// TIA Portal project "GoodBeer_V1" (V16)

(* hardware
DEVICE "Станция S7-1200_1"  S7-1200 Station
   slot 0: "Rack_0"  S7-1200 Rack  Rack  V1.0
   slot 1: "PLC"  CPU 1214C DC/DC/Rly  6ES7 214-1HG40-0XB0  V4.2
   slot 2: "DI 16x24VDC_1"  6ES7 221-1BH32-0XB0  V2.0
   slot 3: "DQ 16xRelay_1"  SM 1222 DQ16 x relay  6ES7 222-1HH32-0XB0  V2.0
   slot 4: "DQ 8xRelay_1"  SM 1222 DQ8 x relay  6ES7 222-1HF32-0XB0  V2.0
   slot 5: "AI 8xRTD_1"  SM 1231 AI8 x RTD  6ES7 231-5PF32-0XB0  V2.0
   slot 6: "AI 8x13 бит_1"  6ES7 231-4HF32-0XB0  V2.0
   slot 7: "AQ 4x14 бит_1"  6ES7 232-4HD32-0XB0  V2.0
   slot 8: "AQ 4x14 бит_2"  6ES7 232-4HD32-0XB0  V2.0
*)

// ===== PLC "PLC"  CPU 1214C DC/DC/Rly =====

VAR_GLOBAL   // PLC tag table "Стандартная таблица переменных"
   "Возврат(1)" AT %M10.6 : Bool;
   "Клавиша Стопа на экране" AT %M202.1 : Bool;
   "клавиша циркуляции" AT %M279.1 : Bool;
   "Циркуляция" AT %M247.2 : Bool;
   "Клапана  в автомат" AT %M38.1 : Bool;
   "mm3" AT %M38.3 : Bool;
   "mm5" AT %M38.4 : Bool;
   "mm6" AT %M38.5 : Bool;
   "mm7" AT %M38.6 : Bool;
   "mm8" AT %M38.7 : Bool;
   "mm9" AT %M39.0 : Bool;
   "mm10" AT %M39.1 : Bool;
   "mm11" AT %M39.2 : Bool;
   "mm12" AT %M39.3 : Bool;
   "mm13" AT %M39.4 : Bool;
   "mm14" AT %M39.5 : Bool;
   "mm15" AT %M39.6 : Bool;
   "mm16" AT %M39.7 : Bool;
   "mm17" AT %M48.2 : Bool;
   "mm18" AT %M48.3 : Bool;
   "mm19" AT %M48.4 : Bool;
   "mm20" AT %M48.5 : Bool;
   "mm21" AT %M48.6 : Bool;
   "mm22" AT %M48.7 : Bool;
   "mm23" AT %M49.0 : Bool;
   "mm24" AT %M49.1 : Bool;
   "mm25" AT %M49.2 : Bool;
   "mm26" AT %M49.3 : Bool;
   "mm27" AT %M49.4 : Bool;
   "mm28" AT %M49.5 : Bool;
   "mm29" AT %M49.6 : Bool;
   "mm30" AT %M49.7 : Bool;
   "mm31" AT %M60.1 : Bool;
   "mm32" AT %M60.2 : Bool;
   "mm33" AT %M60.3 : Bool;
   "mm34" AT %M60.4 : Bool;
   "mm35" AT %M60.5 : Bool;
   "mm36" AT %M60.6 : Bool;
   "mm37" AT %M60.7 : Bool;
   "mm38" AT %M61.0 : Bool;
   "mm39" AT %M61.1 : Bool;
   "mm40" AT %M61.2 : Bool;
   "mm41" AT %M61.3 : Bool;
   "mm42" AT %M61.4 : Bool;
   "mm43" AT %M61.5 : Bool;
   "set1" AT %M61.6 : Bool;
   "set2" AT %M61.7 : Bool;
   "set3" AT %M62.4 : Bool;
   "set4" AT %M62.5 : Bool;
   "ww1" AT %M62.2 : Bool;
   "Косвенное окно1" AT %MB890 : Byte;
   "cw1" AT %M62.3 : Bool;
   "set5" AT %M62.1 : Bool;
   "ww2" AT %M62.0 : Bool;
   "set6" AT %M238.0 : Bool;
   "ww3" AT %M238.1 : Bool;
   "mm4" AT %M238.2 : Bool;
   "set7" AT %M238.3 : Bool;
   "ww4" AT %M238.4 : Bool;
   "set8" AT %M238.5 : Bool;
   "set20" AT %M238.7 : Bool;
   "ww6" AT %M239.0 : Bool;
   "set21" AT %M239.1 : Bool;
   "ww7" AT %M239.2 : Bool;
   "set22" AT %M239.3 : Bool;
   "ww8" AT %M239.4 : Bool;
   "set23" AT %M239.5 : Bool;
   "ww9" AT %M239.6 : Bool;
   "set24" AT %M239.7 : Bool;
   "ww10" AT %M240.0 : Bool;
   "set25" AT %M240.1 : Bool;
   "ww11" AT %M240.2 : Bool;
   "set26" AT %M240.3 : Bool;
   "ww12" AT %M240.4 : Bool;
   "set27" AT %M240.5 : Bool;
   "ww13" AT %M240.6 : Bool;
   "set28" AT %M240.7 : Bool;
   "ww14" AT %M241.0 : Bool;
   "set29" AT %M241.1 : Bool;
   "ww15" AT %M241.2 : Bool;
   "set30" AT %M241.3 : Bool;
   "ww16" AT %M241.4 : Bool;
   "set31" AT %M241.5 : Bool;
   "ww17" AT %M241.6 : Bool;
   "P_Off" AT %M241.7 : Bool;
   "set32" AT %M242.0 : Bool;
   "ww18" AT %M242.1 : Bool;
   "set33" AT %M242.2 : Bool;
   "ww19" AT %M242.3 : Bool;
   "set34" AT %M242.4 : Bool;
   "ww20" AT %M242.5 : Bool;
   "set36" AT %M242.6 : Bool;
   "ww22" AT %M242.7 : Bool;
   "set37" AT %M243.0 : Bool;
   "ww23" AT %M243.1 : Bool;
   "set39" AT %M243.2 : Bool;
   "ww25" AT %M243.3 : Bool;
   "set41" AT %M243.4 : Bool;
   "ww27" AT %M243.5 : Bool;
   "set42" AT %M243.6 : Bool;
   "ww28" AT %M243.7 : Bool;
   "set44" AT %M244.0 : Bool;   // Сообщение при циркуляции
   "ww30" AT %M244.1 : Bool;
   "set51" AT %M244.2 : Bool;
   "ww34" AT %M244.3 : Bool;
   "set61" AT %M244.4 : Bool;
   "ww35" AT %M244.5 : Bool;
   "set53" AT %M244.6 : Bool;
   "ww36" AT %M244.7 : Bool;
   "set54" AT %M245.0 : Bool;
   "ww37" AT %M245.1 : Bool;
   "Вызов экрана аварийный стоп" AT %M245.2 : Bool;
   "косвенное окно2" AT %MB880 : Byte;
   "закрытие окна подтверждения" AT %M245.3 : Bool;
   "Клавиша вытеснение" AT %M104.0 : Bool;
   "Ручная частота насоса M3" AT %MD248 : Real;
   "Бит стерилизации" AT %M245.5 : Bool;
   "Бит выход на режим" AT %M245.6 : Bool;
   "Бит производство" AT %M245.7 : Bool;
   "Бит вытеснения" AT %M247.0 : Bool;
   "Бит мойки" AT %M247.1 : Bool;
   "Tag_30" AT %MD252 : Real;
   "Вкл пида паст" AT %M80.1 : Bool;
   "Выход пид паст %" AT %MW460 : Int;
   "Выход пид произв в %" AT %MW338 : Int;
   "mm2" AT %M11.4 : Bool;
   "mm1" AT %M11.5 : Bool;
   "Выход пид подогрева %" AT %MW362 : Int;
   "Вкл пида охлаждение" AT %M80.2 : Bool;
   "Подтверждение производства" AT %M103.1 : Bool;
   "подтверждение вытеснения" AT %M104.1 : Bool;
   "Обьем выталкивания линий" AT %MD204 : DInt;
   "время процесса в секундах" AT %MD300 : DInt;
   "МИНУТЫ НА ЭКРАН(1)" AT %MD304 : DInt;
   "Время в секундах" AT %MD308 : DInt;
   "СЕКУНДЫ НА ЭКРАН" AT %MD312 : DInt;
   "Информационный бит" AT %MW510 : Int;
   "set40" AT %M24.1 : Bool;
   "ww26" AT %M24.2 : Bool;
   "Нет действий" AT %M110.0 : Bool;
   "Клавиша выхода на режим" AT %M102.0 : Bool;
   "Подтверждение выхода на режим" AT %M102.1 : Bool;
   "Подтверждение мойки" AT %M105.1 : Bool;
   "Готов к производству" AT %M102.7 : Bool;
   "Клавиша производство" AT %M103.0 : Bool;
   "заполнение ок- производство" AT %M103.3 : Bool;
   "Клавиша мойка" AT %M105.0 : Bool;
   "Ополаскивание перед про-ом закончено" AT %M102.3 : Bool;
   "Выход на режим" AT %M102.4 : Bool;
   "Соответствие температур" AT %M279.0 : Bool;
   "Объем заполнения пивом" AT %MD116 : DInt;
   "Tag101" AT %MD120 : DInt;
   "Объем пастеризации" AT %MD124 : DInt;
   "Оъем вытеснения пива" AT %MD128 : DInt;
   "Tag104" AT %MD132 : DInt;
   "Tag105" AT %MD136 : Real;
   "Tag106" AT %MD140 : Real;
   "Tag107" AT %MD144 : DInt;
   "Tag108" AT %MD148 : DInt;   // Соощение при переходе на циркуляцию по температуре
   "Расчетная ПЕ температура" AT %MD70 : Real;
   "tag71" AT %MD74 : Real;
   "tag72" AT %MD82 : Time;
   "tag73" AT %MD86 : Real;
   "tag74" AT %MD90 : Real;
   "tag75" AT %MD94 : Time;
   "Заполнение пастеризатора пивом, вытеснение воды" AT %M103.2 : Bool;
   "Текущий объем заполнения" AT %MD504 : DInt;
   "Счетчик производства" AT %MD508 : DInt;
   "Вытеснение пива в буфер" AT %M104.2 : Bool;
   "Объем вытеснения" AT %MW104 : Int;
   "Вытеснение ок" AT %M104.3 : Bool;
   "Ополаскивание после производства" AT %M104.4 : Bool;
   "Ополаскивание ок" AT %M104.5 : Bool;
   "Производство" AT %M103.4 : Bool;
   "Вкл пида производительности" AT %M80.3 : Bool;
   "Режим СIP вкл" AT %M105.2 : Bool;
   "Время ополаскивания" AT %MD0 : Time;
   "flag" AT %M5.3 : Bool;
   "flag1" AT %M5.4 : Bool;
   "flag2" AT %M5.5 : Bool;
   "flag3" AT %M5.6 : Bool;
   "flag4" AT %M5.7 : Bool;
   "flag5" AT %M6.0 : Bool;
   "flag6" AT %M6.1 : Bool;
   "flag7" AT %M6.2 : Bool;
   "flag8" AT %M6.3 : Bool;
   "flag9" AT %M6.4 : Bool;
   "flag10" AT %M6.5 : Bool;
   "flag11" AT %M6.6 : Bool;
   "flag12" AT %M6.7 : Bool;
   "flag13" AT %M7.0 : Bool;
   "flag14" AT %M7.1 : Bool;
   "flag15" AT %M7.2 : Bool;
   "flag16" AT %M7.3 : Bool;
   "flag17" AT %M7.4 : Bool;
   "flag18" AT %M7.5 : Bool;
   "flag19" AT %M7.6 : Bool;
   "flag20" AT %M7.7 : Bool;
   "flag21" AT %M8.0 : Bool;
   "flag22" AT %M8.1 : Bool;
   "flag23" AT %M8.2 : Bool;
   "flag24" AT %M8.3 : Bool;
   "flag25" AT %M8.4 : Bool;   // НЕт расхода при мойке СИП
   "Розлив" AT %M9.1 : Bool;
   "Мойка" AT %M9.2 : Bool;
   "Флип1" AT %M9.3 : Bool;
   "Флип11" AT %M9.4 : Bool;
   "Флип2" AT %M9.5 : Bool;
   "Флип22" AT %M9.6 : Bool;
   "Откачка" AT %M9.7 : Bool;
   "Подтверждение включения нагрева" AT %M102.5 : Bool;
   "Оъем воды Ополаскивания" AT %MD190 : DInt;
   "Ополаскивание по счетчику" AT %M10.5 : Bool;   // выбор типа отсчета режима опаласкивания 1 - по счетчику 0 - по времени
   "Мин_УстВрЦиркул" AT %MD12 : DInt;   // Время циркуляции до аварии в мин
   "ВремяВРежимеЦиркул" AT %MD16 : DInt;
   "flag26" AT %M11.3 : Bool;
   "Вкл Регулятора давления" AT %M11.6 : Bool;
   "Отключить_Не использую" AT %M11.7 : Bool;   // Отключаю не нужную ветку
   "Время в циркуляции" AT %MD44 : Time;   // Время пройденной с момента циркуляции
   "Стоп циркул" AT %M24.0 : Bool;
   "Вкл пида нагрев Мойка" AT %M48.0 : Bool;
   "Уставка нагревателя" AT %MD164 : Real;
   "flag27" AT %M63.0 : Bool;
   "НетПотокМойкаВнутр" AT %M63.2 : Bool;
   "НетПотокМойкаВнешняя" AT %M63.3 : Bool;
END_VAR

VAR_GLOBAL   // PLC tag table "AI"
   "AI Тем. вых. пива" AT %IW112 : Int;
   "AI Тем. Пропиленгликоль" AT %IW114 : Int;
   "AI Тем. Регенерации" AT %IW116 : Int;
   "AI Тем. Пастеризации" AT %IW118 : Int;
   "AI Тем. ГВ пастеризации" AT %IW120 : Int;
   "AI Давл. Пастеризация" AT %IW122 : Int;
   "AI Тем. в буфере" AT %IW124 : Int;
   "AI Давл. на розлив" AT %IW126 : Int;
   "AI Расходомер" AT %IW128 : Int;
   "AI1" AT %IW130 : Int;
   "AI2" AT %IW132 : Int;
   "AI3" AT %IW134 : Int;
   "AQ Насос продукта" AT %QW128 : Int;
   "AQ Насос бустерный" AT %QW130 : Int;
   "AQ Насос розлива" AT %QW144 : Int;
   "AQ Пропиленгликоль" AT %QW146 : Int;
   "AQ  Пар" AT %QW148 : Int;
   "AQ" AT %QW150 : Int;
   "Тем. Входа пропиленгликоль" AT %MD250 : Real;
   "Тем. Входа с регенерации" AT %MD254 : Real;
   "Тем. Пастеризации" AT %MD258 : Real;
   "Тем. контура ГВ" AT %MD262 : Real;
   "Тем. в буфере" AT %MD266 : Real;
   "Давление розлив" AT %MD270 : Real;
   "Расход ПОУ" AT %MD274 : Real;
   "Заполнение пастеризатора водой" AT %M278.0 : Bool;
   "Время заполнения пастеризатора" AT %MD280 : Time;
   "Давление пастеризации" AT %MD284 : Real;
   "Тем. Выхода пива" AT %MD288 : Real;
   "AI TT1" AT %IW150 : Int;   // Темп входа пива PT100
   "AI TT2" AT %IW152 : Int;   // Темп выхода пива PT100
   "AI TT3" AT %IW154 : Int;   // Темп ГВ - нагрев PT100
   "AI TT4" AT %IW156 : Int;   // Темп Гликоль PT100
   "AI TT5" AT %IW158 : Int;   // ТЕмп емкость PT100
   "AI TT6" AT %IW184 : Int;   // Темп выход продукт ТТ6 4-20 мА
   "AI Расходомерр" AT %IW170 : Int;   // Расходомер 4-20
   "AI PT1" AT %IW172 : Int;   // Датчик давления 4-20
   "AI PT2 - Секция пастеризации" AT %IW174 : Int;   // Датчик давления 4-20
   "AI PT3" AT %IW176 : Int;   // Датчик давления 4-20
   "AI WT" AT %IW178 : Int;   // Датчик веса буфера
   "AI CT" AT %IW182 : Int;   // Датчик концентрации
END_VAR

VAR_GLOBAL   // PLC tag table "DI"
   "Реле давл. воздуха" AT %I0.7 : Bool;
   "Импульс с расходомера" AT %I2.6 : Bool;
   "Автомат QF1" AT %I19.4 : Bool;
   "Автомат QF2" AT %I19.5 : Bool;
   "Автомат QF3" AT %I19.6 : Bool;
   "Автомат QF4" AT %I19.7 : Bool;
   "Автомат QF5" AT %I20.0 : Bool;
   "DI1" AT %I20.1 : Bool;
   "DI2" AT %I20.2 : Bool;
   "ZP1" AT %I20.3 : Bool;
   "ZP2" AT %I20.4 : Bool;
   "ZP3" AT %I20.5 : Bool;
   "ZP4" AT %I20.6 : Bool;
   "ZP5" AT %I20.7 : Bool;
   "ZP6" AT %I21.0 : Bool;
   "ZP7" AT %I21.1 : Bool;
   "ZP8" AT %I21.2 : Bool;
   "ZP9" AT %I21.3 : Bool;
   "Аварийный STOP" AT %I0.0 : Bool;
   "Реле обрыв/перекос фазы" AT %I0.1 : Bool;
   "Работа ПЧ-1" AT %I0.2 : Bool;
   "Работа ПЧ-2" AT %I0.3 : Bool;
   "Работа ПЧ-3" AT %I0.4 : Bool;
   "Работа ПЧ-4" AT %I0.5 : Bool;
   "Работа ПЧ-5" AT %I0.6 : Bool;
   "Состояние V1" AT %I1.0 : Bool;
   "Состояние V2" AT %I1.1 : Bool;
   "Состояние V3" AT %I10.2 : Bool;
   "Состояние V4" AT %I1.2 : Bool;
   "Состояние V5" AT %I1.3 : Bool;
   "Состояние V6" AT %I1.4 : Bool;
   "Состояние V7" AT %I1.5 : Bool;
   "Состояние V8" AT %I2.0 : Bool;
   "Состояние V9" AT %I2.1 : Bool;
   "Состояние V10" AT %I2.2 : Bool;
   "LS1 - Низ Буфер" AT %I2.3 : Bool;
   "LS2 - Верх Буфер" AT %I2.4 : Bool;
   "LS3 - Латерн" AT %I2.5 : Bool;
   "Калач ZS1" AT %I3.0 : Bool;
   "Калач ZS2" AT %I3.1 : Bool;
   "Калач ZS3" AT %I3.2 : Bool;
   "Калач ZS4" AT %I3.3 : Bool;
   "Калач ZS5" AT %I3.4 : Bool;
   "Калач ZS6" AT %I3.5 : Bool;
   "Калач ZS7" AT %I3.6 : Bool;
END_VAR

VAR_GLOBAL   // PLC tag table "Пневмоостров"
   "Подпитка воды КО1" AT %Q20.0 : Bool;
   "Пар отсечной КО2" AT %Q20.1 : Bool;
   "Вход пива ZP8" AT %Q20.2 : Bool;
   "NLS давление" AT %Q20.3 : Bool;
   "Вход сетевой воды ZP7" AT %Q20.4 : Bool;
   "Вход пропиленгликоль ZP9" AT %Q20.5 : Bool;
   "Байпас емкость ZP2" AT %Q20.6 : Bool;
   "Трап ZP3" AT %Q20.7 : Bool;
   "Заполнение ZP5" AT %Q21.0 : Bool;
   "Розлив ZP1" AT %Q21.1 : Bool;
   "МГ буфер ZP6" AT %Q21.2 : Bool;
   "Циркуляция ZP4" AT %Q21.3 : Bool;
   "13" AT %Q21.4 : Bool;
   "14" AT %Q21.5 : Bool;
   "Кл Возврата ZP6" AT %Q21.6 : Bool;
END_VAR

VAR_GLOBAL   // PLC tag table "Аварии"
   "Авария клапана ZP8" AT %M4.0 : Bool;
   "Авария клапана ZP7" AT %M4.1 : Bool;
   "Авария клапана ZP9" AT %M4.2 : Bool;
   "Авария клапана ZP2" AT %M4.3 : Bool;
   "Авария клапана ZP3" AT %M4.4 : Bool;
   "Авария клапана ZP5" AT %M4.5 : Bool;
   "Авария клапана ZP6" AT %M4.6 : Bool;
   "Авария клапана ZP4" AT %M4.7 : Bool;
   "Авария клапана ZP1" AT %M5.0 : Bool;
   "Авария давления воздуха" AT %M5.1 : Bool;
   "Реле 380V" AT %M5.2 : Bool;
   "Включение звука" AT %M8.5 : Bool;
   "Клавиша сброса звука" AT %M8.6 : Bool;
   "Задержка насоса" AT %M8.7 : Bool;
   "Авария низкий расход" AT %M9.0 : Bool;
   "Авария M1" AT %M10.0 : Bool;
   "Авария М2" AT %M10.1 : Bool;
   "Авария М3" AT %M10.2 : Bool;
   "Авария М5" AT %M10.3 : Bool;
   "Авария М4" AT %M10.4 : Bool;
   "Авария давления секции пастеризации" AT %M247.5 : Bool;
   "Авария ГВ контур паст" AT %M247.3 : Bool;
   "Аварийная остановка" AT %M202.0 : Bool;
   "Циркул_Долгая_Сигнал" AT %M10.7 : Bool;   // Сигнал о длительной циркуляции
END_VAR

VAR_GLOBAL   // PLC tag table "DO"
   "Зеленый" AT %Q5.5 : Bool;
   "Красный" AT %Q5.3 : Bool;
   "Сирена" AT %Q5.6 : Bool;
   "Желтый" AT %Q5.4 : Bool;
   "Насос М1" AT %Q3.0 : Bool;   // Продукт
   "Насос М2" AT %Q3.1 : Bool;   // Продукт - 2
   "Насос М3" AT %Q3.2 : Bool;   // Продукт из Буфера
   "Насос М4" AT %Q3.3 : Bool;   // Теплоноситель
   "Насос М5" AT %Q3.4 : Bool;   // Хладоген
   "V1_Вода" AT %Q0.0 : Bool;
   "V2_Продукт" AT %Q0.1 : Bool;
   "V3_Давления" AT %Q0.2 : Bool;
   "V4_Циркуляция" AT %Q0.3 : Bool;
   "V5_Дренаж (НО)" AT %Q0.4 : Bool;
   "V6_Возврат" AT %Q0.5 : Bool;
   "V7_Моющая головка" AT %Q0.6 : Bool;
   "V8_Вход пр в бочку" AT %Q0.7 : Bool;
   "V9_Выход пр из бочки" AT %Q1.0 : Bool;
   "V10_клапан" AT %Q1.1 : Bool;
   "V11_Запорный тепло" AT %Q4.0 : Bool;
   "V12_Запор гликоль" AT %Q4.1 : Bool;
   "V13_Сброс дав емкость" AT %Q4.2 : Bool;
   "V14_Щелочь" AT %Q4.3 : Bool;
   "V16_Кислота" AT %Q4.5 : Bool;
   "V15_Насос Щелочь" AT %Q4.4 : Bool;
   "V17_Насос Кислота" AT %Q4.6 : Bool;
END_VAR

VAR_GLOBAL   // PLC tag table "AO"
   "AO Скорость M1" AT %QW190 : Int;
   "AO Скорость M2" AT %QW192 : Int;
   "AO Скорость M3" AT %QW194 : Int;
   "AO Скорость M4" AT %QW196 : Int;
   "AO Скорость M5" AT %QW198 : Int;
   "AO V11.1" AT %QW200 : Int;   // Клапан Нагрева
   "AO V12.1" AT %QW202 : Int;   // Клапан Охлаждения
   "AO V3 (NO)" AT %QW204 : Int;   // Клапан регул давления (100-0) инверсия
END_VAR

VAR_GLOBAL   // PLC tag table "Timers_CPU"
   "Time_0.1s" AT %M500.0 : Bool;
   "Time_0.2s" AT %M500.1 : Bool;
   "Time_0.4s" AT %M500.2 : Bool;
   "Time_0.5s" AT %M500.3 : Bool;
   "Time_0.8s" AT %M500.4 : Bool;
   "Time_1s" AT %M500.5 : Bool;
   "Time_1.6s" AT %M500.6 : Bool;
   "Time_2s" AT %M500.7 : Bool;
END_VAR

VAR_GLOBAL   // PLC tag table "_test"
   "tInValue" AT %MW20 : Int;
   "tTypeSens" AT %MW22 : Int;
   "tEn_Sin" AT %M11.0 : Bool;
   "tSim_value" AT %MD26 : Real;
   "tLL" AT %MD30 : Real;
   "tHH" AT %MD34 : Real;
   "tFilter" AT %M11.1 : Bool;
   "BlinkForExhibition" AT %M24.3 : Bool;   // временный для мигания лампочки на выстовке
   "Test_1_IN" AT %M24.4 : Bool;
   "Test_1_Out" AT %M24.5 : Bool;
   "Test_2_IN" AT %M24.6 : Bool;
   "Test_2_Out" AT %M24.7 : Bool;
   "t_Start_Wash" AT %M25.0 : Bool;
   "t_Stop_Wash" AT %M25.1 : Bool;
   "t_Ch_Alkai" AT %M25.2 : Bool;
   "t_Ch_Acid" AT %M25.3 : Bool;
   "t_LS2" AT %M25.4 : Bool;
   "t_LS_1" AT %M25.5 : Bool;
   "t_Flow_Ok" AT %M25.6 : Bool;
   "t_Water_Count" AT %M25.7 : Bool;
   "t_Conc_Act" AT %MD50 : Real;
   "t_Conc_Set" AT %MD54 : Real;
   "t_ConcDelta" AT %MD64 : Real;
   "t_TempActual" AT %MD98 : Real;
   "t_TempSet" AT %MD112 : Real;
   "t_ALARM" AT %M38.0 : Bool;
   "T_WashActive" AT %M38.2 : Bool;
   "tdeltaTemp" AT %MD158 : Real;
   "nextStep" AT %M78.0 : Bool;
END_VAR

VAR_GLOBAL   // PLC tag table "Тэги для HMI"
   "fb_AI_Темп входа пива PT100" AT %MD400 : Real;   // Обработанный сигнал с датчика
   "fb_AI_Темп выхода пива  PT100" AT %MD404 : Real;   // Обработанный сигнал с датчика
   "fb_AI_Темп ГВ - нагрев PT100" AT %MD408 : Real;   // Обработанный сигнал с датчика
   "fb_AI_Темп Гликоль PT100" AT %MD412 : Real;   // Обработанный сигнал с датчика
   "fb_AI_ТЕмп емкость PT100" AT %MD416 : Real;   // Обработанный сигнал с датчика
   "fb_AI_Темп выход продукт ТТ6 4-20 мА" AT %MD420 : Real;   // Обработанный сигнал с датчика
   "fb_AI_Расходомер 4-20" AT %MD424 : Real;   // Обработанный сигнал с датчика
   "fb_AI_M2_давления 4-20" AT %MD428 : Real;   // Обработанный сигнал с датчика
   "fb_AI_Выход пива давления 4-20" AT %MD432 : Real;   // Обработанный сигнал с датчика
   "fb_AI_Выход Буфера давления 4-20" AT %MD436 : Real;   // Обработанный сигнал с датчика
   "fb_AI_Датчик веса буфера" AT %MD440 : Real;   // Обработанный сигнал с датчика
   "fb_AI_Датчик концентрации" AT %MD444 : Real;   // Обработанный сигнал с датчика
   "fb_DI_Аварийный STOP" AT %M448.0 : Bool;   // Обработанный сигнал DI
   "fb_DI_Реле обрыв/перекос фазы" AT %M448.1 : Bool;   // Обработанный сигнал DI
   "fb_DI_Работа ПЧ-1" AT %M448.2 : Bool;   // Обработанный сигнал DI
   "fb_DI_Работа ПЧ-2" AT %M448.3 : Bool;   // Обработанный сигнал DI
   "fb_DI_Работа ПЧ-3" AT %M448.4 : Bool;   // Обработанный сигнал DI
   "fb_DI_Работа ПЧ-4" AT %M448.5 : Bool;   // Обработанный сигнал DI
   "fb_DI_Работа ПЧ-5" AT %M448.6 : Bool;   // Обработанный сигнал DI
   "fb_DI_Реле давл. воздуха" AT %M448.7 : Bool;   // Обработанный сигнал DI
   "fb_DI_Состояние V1" AT %M449.0 : Bool;   // Обработанный сигнал DI
   "fb_DI_Состояние V2" AT %M449.1 : Bool;   // Обработанный сигнал DI
   "fb_DI_Состояние V3" AT %M449.2 : Bool;   // Обработанный сигнал DI
   "fb_DI_Состояние V4" AT %M449.3 : Bool;   // Обработанный сигнал DI
   "fb_DI_Состояние V5" AT %M449.4 : Bool;   // Обработанный сигнал DI
   "fb_DI_Состояние V6" AT %M449.5 : Bool;   // Обработанный сигнал DI
   "fb_DI_Состояние V7" AT %M449.6 : Bool;   // Обработанный сигнал DI
   "fb_DI_Состояние V8" AT %M449.7 : Bool;   // Обработанный сигнал DI
   "fb_DI_Состояние V9" AT %M450.0 : Bool;   // Обработанный сигнал DI
   "fb_DI_Состояние V10" AT %M450.1 : Bool;   // Обработанный сигнал DI
   "fb_DI_LS1 - Низ Буфер" AT %M450.2 : Bool;   // Обработанный сигнал DI
   "fb_DI_LS2 - Верх Буфер" AT %M450.3 : Bool;   // Обработанный сигнал DI
   "fb_DI_LS3 - Латерн" AT %M450.4 : Bool;   // Обработанный сигнал DI
   "fb_DI_Импульс с расходомера" AT %M450.5 : Bool;   // Обработанный сигнал DI
   "fb_DI_Калач ZS1" AT %M450.6 : Bool;   // Обработанный сигнал DI
   "fb_DI_Калач ZS2" AT %M450.7 : Bool;   // Обработанный сигнал DI
   "fb_DI_Калач ZS3" AT %M451.0 : Bool;   // Обработанный сигнал DI
   "fb_DI_Калач ZS4" AT %M451.1 : Bool;   // Обработанный сигнал DI
   "fb_DI_Калач ZS5" AT %M451.2 : Bool;   // Обработанный сигнал DI
   "fb_DI_Калач ZS6" AT %M451.3 : Bool;   // Обработанный сигнал DI
   "fb_DI_Калач ZS7" AT %M451.4 : Bool;   // Обработанный сигнал DI
   "fb_DI_Калач ZS8" AT %M451.5 : Bool;   // Обработанный сигнал DI
   "bHMI_ResetAlarm" AT %M11.2 : Bool;   // Сброс Аварий
   "bmAlarm" AT %M80.0 : Bool;   // main ALARM
   "iPID_Out_Нагрев" AT %MW680 : Int;   // Выход из ПИД Нагрев
   "iPID_Out_Гликоль" AT %MW682 : Int;   // Выход из ПИД охлаждение
   "iPID_Out_Кл.Давления" AT %MW684 : Int;   // Выход из ПИД Давлеие
   "iPid_Out_Насос продукта-1" AT %MW698 : Int;
   "iPid_Out_Насос продукта-2" AT %MW700 : Int;
   "rCalculate_PE_from_Te" AT %MD106 : Real;   // Расчетное значение ПЕ получаемое после ввода температуры
   "PE_Fact" AT %MD40 : Real;
   "iTime_Min_Wash" AT %MW152 : Int;   // Минуты для дисплея в режиме мойка
   "iTime_Sec_Wash" AT %MW156 : Int;   // Сек для дисплея в режиме мойка
   "bWash_In_Work" AT %M162.0 : Bool;   // Статус работа внутренней мойки
   "iStepWash" AT %MW58 : Int;   // Шаг мойки
   "iCounterWash" AT %MW68 : Int;   // Счетчик воды в режиме мойка
   "bStart_Wash" AT %M60.0 : Bool;   // Старт Мойки
   "b_Выбор_Щелочь" AT %M62.6 : Bool;   // Выбор мойки с щелочью
   "b_Выбор-Кислота" AT %M48.1 : Bool;   // Выбор мойки с кислотой
   "bAllAuto" AT %M62.7 : Bool;   // Все в автомат
   "bMessage_Temp_Cirkil" AT %M63.1 : Bool;   // Сообщение отклонение температуры - переход в циркуляцию
END_VAR

TYPE "ty_DI"
   STRUCT
      In : Bool;
      Sim : Bool;
      Sim_Out : Bool;
      Filtr : Bool;
      TimeFiltr : DInt;
      Out : Bool;
   END_STRUCT;
END_TYPE

TYPE "ty_Pump"
   STRUCT
      bManualMode : Bool;   // Выбор рунчого режима
      bManualStart : Bool;   // Старт/Стоп в ручном режиме
      rManualSpeed : Real;   // СКрорсть в ручном режиме
      bAutoCMD : Bool;   // Команда в автоматическом режиме
      rAutoSpeed : Real;   // Скорость в автомате
      bHMI_RUN_State : Bool;   // Статус Работа/стоп для HMI
      "rHMI_Speed%" : Real;   // Скорость насоса в % для HMI
      bResAlarm : Bool;   // Сброс аварии насоса
      bALARM : Bool;   // АвАрия насоса
      iHMI_Status : Int;   // Статус для HMII
   END_STRUCT;
END_TYPE

TYPE "ty_AI"
   STRUCT
      iTypeSensor : Int;   // 0 - 4-20 $ 1 - RTD Тип датчика
      bSimEnable : Bool;   // Вкл СИМУЛЯЦИЯ
      rSimValue : Real;   // Значение симул
      rHL : Real;   // Нижний предел датчика
      rLL : Real;   // Верхний предел датчика
      bFilterEnable : Bool;   // Включение фильтрации
      rOut_Value : Real;   // Выходное значение
      bOut_Error : Bool;   // Выход ошибки
   END_STRUCT;
END_TYPE

TYPE "ty_Valve"
   STRUCT
      bManualMode : Bool;   // входы
      bManualOpen : Bool;   // входы
      bAuto_OpenCmd : Bool;   // входы
      bHaveFeedback : Bool;   // входы
      bFeedbackOpen : Bool;   // входы
      bResetAlarm : Bool;   // входы
      tMaxTime : DInt := 100;   // входы
      bValveOut : Bool;   // Выходы
      bValveFault : Bool;   // Выходы
      iValveState : Int;   // Выходы
   END_STRUCT;
END_TYPE

TYPE "ty_Valve-regul"
   STRUCT
      bManualMode : Bool;   // Переключение режима
      rManualSetpoint : Real;   // Ручной режим - уствка
      bManualOpenClose : Bool;   // Ручной реж - откр/закрыть
      bAutoOpenClose : Bool;   // Автомат открыть/закрыть
      rAutoSetpoint : Real;   // Автомат значение
      bOut_OpenClose : Bool;   // Выход Открыть/зактрыть
      iAnalogOutput : Int;   // Выход Аналог значение
      rValvePosPercent : Real;   // Выход для HMI
      bStatusValveOpen : Bool;   // Выход для статуса HMI
   END_STRUCT;
END_TYPE

DATA_BLOCK "Уставки"   // DB2
{ S7_Optimized_Access := 'FALSE' }
VERSION : 0.1
   VAR
      "Ручная уставка насос ГВ подогрева" : Int := 0;
      "Ручная частота насоса ГВ паст" : Int := 0;
      "Уставка Т паст" : Real := 0.0;
      "Уставки Т подогрев" : Real := 2.0;   // ТЕмпература выхода пива после охлаждения
      "Уставки давления" : Real;
      "Уставка расхода" : Real := 2.0;
      "Уставка расхода_М3" : Real;   // Уставка расхода насоса М3
      "Уставка давления выхода" : Real := 1.5;
      "Ручная частота насоса M1" : Int := 100;
      "Ручная частота насоса M2" : Int := 100;
      "Ручная частота насоса M5" : Int := 80;
      "Уставка аварии перегрева" : Real := 0.0;
      "Уставка ПЕ" : Real := 540.0;
      "Значение для аварии циркуляции" : Real := 5.0;
      "Погрешность температуры пастеризации" : Real := 3.0;
      "Погрешность температуры выхода" : Real := 6.0;
      "Аварийное давление" : Real := 15.0;
      "Выбор уставки для пастеризации" : Bool;   // 0 - вводится уставка ПЕ, 1 - вводится желаемая температура
      "Уставка темп пастеризации" : Real;   // Если выбран ввод уставки по температуре то вводить желаемую уставку
      "Минимальный расход - Авария" : Real := 0.1;   // Минимальный расход - Авария
      "Авар Темп контур ГВ" : Real := 100.0;   // аварийная темп контура ГВ
   END_VAR
BEGIN
END_DATA_BLOCK

DATA_BLOCK "Параметры"   // DB5
{ S7_Optimized_Access := 'FALSE' }
VERSION : 0.1
   VAR
      "Время ополаскивания перед выходом на режим" : Int := 3;
      "Время ополаскивания после производства" : Int := 2;
      "Время циркуляции до аварии" : Int;   // мин
      "Производительность при мойке" : Real := 4.0;
      "Обьем заполнения пастеризатора пивом" : Int := 105;
      "Объем вытеснения пива водой" : Int := 85;
      "Объем воды Ополаскивания" : Int := 10;
      LS2_ChoosWhatDo_FlushOrCirculate : Bool;   // 1 - Выталкив/0- Циркул - что делаем при сработке LS2 циркуляция или выталкивание
      bНасос_М3_РаботаПоПИД : Bool;   // 1 - ПИД 0- Уставка скорости
   END_VAR
BEGIN
END_DATA_BLOCK

DATA_BLOCK "Уставки_Мойка_Вн"   // DB19
{ S7_Optimized_Access := 'FALSE' }
VERSION : 0.1
   VAR
      iCount_Water_Наполнение : Int := 10;   // Уставка счетчика наполнения
      iCount_Water_ПолосЩелочи : Int := 10;   // Уставка счетчика ополаскивания после щелочи
      iCount_Water_ПолосКислоты : Int := 10;   // Уставка счетчика ополаскивания после Кислоты
      "dwВремяФлипованияКл,сек" : DInt := 3;   // сек, Время переключения клапанов - Флипование
      "dwВремяПаузыФлипованияКл,сек_1" : DInt;   // сек, Время паузы - Флипование
      "dwВремяЦиркуляции,мин" : DInt := 1;   // мин, время циркуляции
      "dwВремяЩОЛОЧЬ_Циркул,ми" : DInt := 5;   // мин, время циркуляции ЩЕЛОЧИ
      "dwВремяКислота_Циркул,ми" : DInt := 5;   // мин, время циркуляции Кислота
      dwВремяИмпНаведения : DInt := 2;   // сек, Время продолжительности добавления химии
      dwПаузыИмпНаведения : DInt := 30;   // сек, Вермя паузы между порциями химии
      rSet_Concentr_Щелочь : DInt := 2000;   // Уставка концентрата щелочи
      rSet_Concentr_Кислота : DInt := 5000;   // Уставка концентрата Кислоты
      rSet_Concentr_Вода : DInt := 100;   // Уставка концентрата Вода
      rSet_Conc_Delta : DInt := 50;   // Дельта отклонения от уставки
      rSet_Temp_Nagrev_Wash : Real := 50.0;   // Уставка нагрева для мойки ПИД
      rSet_Temp_Nagrev_Вода : Real;
      rSet_Temp_Nagrev_Щелочь : Real;
      rSet_Temp_Nagrev_Кислота : Real;
      rSet_Delta_Temp : Real := 5.0;   // Дельта температуры нагрева
   END_VAR
BEGIN
END_DATA_BLOCK

DATA_BLOCK "Флипование_DB"   // DB54
{ S7_Optimized_Access := 'TRUE' }
VERSION : 0.1
// stored: InstanceOfName Флипование
"Флипование"
BEGIN
END_DATA_BLOCK

// folder: AI/DB

DATA_BLOCK "AI_Univ_DB_9"   // DB40
{ S7_Optimized_Access := 'TRUE' }
VERSION : 0.1
// stored: InstanceOfName AI_Univ
"AI_Univ"
BEGIN
END_DATA_BLOCK

DATA_BLOCK "AI_Univ_DB_6"   // DB41
{ S7_Optimized_Access := 'TRUE' }
VERSION : 0.1
// stored: InstanceOfName AI_Univ
"AI_Univ"
BEGIN
END_DATA_BLOCK

DATA_BLOCK "AI_Univ_DB_5"   // DB42
{ S7_Optimized_Access := 'TRUE' }
VERSION : 0.1
// stored: InstanceOfName AI_Univ
"AI_Univ"
BEGIN
END_DATA_BLOCK

DATA_BLOCK "AI_Univ_DB_4"   // DB43
{ S7_Optimized_Access := 'TRUE' }
VERSION : 0.1
// stored: InstanceOfName AI_Univ
"AI_Univ"
BEGIN
END_DATA_BLOCK

DATA_BLOCK "AI_Univ_DB_3"   // DB44
{ S7_Optimized_Access := 'TRUE' }
VERSION : 0.1
// stored: InstanceOfName AI_Univ
"AI_Univ"
BEGIN
END_DATA_BLOCK

DATA_BLOCK "AI_Univ_DB_8"   // DB45
{ S7_Optimized_Access := 'TRUE' }
VERSION : 0.1
// stored: InstanceOfName AI_Univ
"AI_Univ"
BEGIN
END_DATA_BLOCK

DATA_BLOCK "AI_Univ_DB_1"   // DB46
{ S7_Optimized_Access := 'TRUE' }
VERSION : 0.1
// stored: InstanceOfName AI_Univ
"AI_Univ"
BEGIN
END_DATA_BLOCK

DATA_BLOCK "AI_Univ_DB_2"   // DB47
{ S7_Optimized_Access := 'TRUE' }
VERSION : 0.1
// stored: InstanceOfName AI_Univ
"AI_Univ"
BEGIN
END_DATA_BLOCK

DATA_BLOCK "AI_Univ_DB_7"   // DB48
{ S7_Optimized_Access := 'TRUE' }
VERSION : 0.1
// stored: InstanceOfName AI_Univ
"AI_Univ"
BEGIN
END_DATA_BLOCK

DATA_BLOCK "AI_Univ_DB_10"   // DB49
{ S7_Optimized_Access := 'TRUE' }
VERSION : 0.1
// stored: InstanceOfName AI_Univ
"AI_Univ"
BEGIN
END_DATA_BLOCK

DATA_BLOCK "AI_Univ_DB_12"   // DB50
{ S7_Optimized_Access := 'TRUE' }
VERSION : 0.1
// stored: InstanceOfName AI_Univ
"AI_Univ"
BEGIN
END_DATA_BLOCK

DATA_BLOCK "AI_Univ_DB_11"   // DB51
{ S7_Optimized_Access := 'TRUE' }
VERSION : 0.1
// stored: InstanceOfName AI_Univ
"AI_Univ"
BEGIN
END_DATA_BLOCK

// folder: DI

DATA_BLOCK "DI_fb_Arrey_DB"   // DB30
{ S7_Optimized_Access := 'TRUE' }
VERSION : 0.1
// stored: InstanceOfName DI_fb_Arrey
"DI_fb_Arrey"
BEGIN
END_DATA_BLOCK

DATA_BLOCK "DI_fb_Arrey_Old_DB"   // DB37
{ S7_Optimized_Access := 'TRUE' }
VERSION : 0.1
// stored: InstanceOfName DI_fb_Arrey_Old
"DI_fb_Arrey_Old"
BEGIN
END_DATA_BLOCK

// folder: Pumps

DATA_BLOCK "FB_Pump_DB_1"   // DB29
{ S7_Optimized_Access := 'FALSE' }
VERSION : 0.1
// stored: InstanceOfName FB_Pump
"FB_Pump"
BEGIN
END_DATA_BLOCK

DATA_BLOCK "FB_Pump_DB_2"   // DB33
{ S7_Optimized_Access := 'FALSE' }
VERSION : 0.1
// stored: InstanceOfName FB_Pump
"FB_Pump"
BEGIN
END_DATA_BLOCK

DATA_BLOCK "FB_Pump_DB_3"   // DB34
{ S7_Optimized_Access := 'FALSE' }
VERSION : 0.1
// stored: InstanceOfName FB_Pump
"FB_Pump"
BEGIN
END_DATA_BLOCK

DATA_BLOCK "FB_Pump_DB_5"   // DB35
{ S7_Optimized_Access := 'FALSE' }
VERSION : 0.1
// stored: InstanceOfName FB_Pump
"FB_Pump"
BEGIN
END_DATA_BLOCK

DATA_BLOCK "FB_Pump_DB_4"   // DB36
{ S7_Optimized_Access := 'FALSE' }
VERSION : 0.1
// stored: InstanceOfName FB_Pump
"FB_Pump"
BEGIN
END_DATA_BLOCK

// folder: System blocks/Program resources

DATA_BLOCK "IEC_Timer_0_DB"   // DB6
{ S7_Optimized_Access := 'TRUE' }
AUTHOR : Simatic
FAMILY : IEC
NAME : IEC_TMR
VERSION : 1.0
// stored: InstanceOfName IEC_TIMER
"IEC_TIMER"
BEGIN
END_DATA_BLOCK

DATA_BLOCK "IEC_Timer_0_DB_1"   // DB7
{ S7_Optimized_Access := 'TRUE' }
AUTHOR : Simatic
FAMILY : IEC
NAME : IEC_TMR
VERSION : 1.0
// stored: InstanceOfName IEC_TIMER
"IEC_TIMER"
BEGIN
END_DATA_BLOCK

DATA_BLOCK "IEC_Counter_0_DB"   // DB8
{ S7_Optimized_Access := 'TRUE' }
AUTHOR : SIMATIC
FAMILY : IEC
NAME : DCNTR
VERSION : 1.2
// stored: InstanceOfName IEC_DCOUNTER
"IEC_DCOUNTER"
BEGIN
END_DATA_BLOCK

DATA_BLOCK "IEC_Counter_0_DB_1"   // DB9
{ S7_Optimized_Access := 'TRUE' }
AUTHOR : SIMATIC
FAMILY : IEC
NAME : DCNTR
VERSION : 1.2
// stored: InstanceOfName IEC_DCOUNTER
"IEC_DCOUNTER"
BEGIN
END_DATA_BLOCK

DATA_BLOCK "IEC_Counter_0_DB_2"   // DB10
{ S7_Optimized_Access := 'TRUE' }
AUTHOR : SIMATIC
FAMILY : IEC
NAME : DCNTR
VERSION : 1.2
// stored: InstanceOfName IEC_DCOUNTER
"IEC_DCOUNTER"
BEGIN
END_DATA_BLOCK

DATA_BLOCK "IEC_Timer_0_DB_2"   // DB11
{ S7_Optimized_Access := 'TRUE' }
AUTHOR : Simatic
FAMILY : IEC
NAME : IEC_TMR
VERSION : 1.0
// stored: InstanceOfName IEC_TIMER
"IEC_TIMER"
BEGIN
END_DATA_BLOCK

DATA_BLOCK "IEC_Timer_0_DB_3"   // DB12
{ S7_Optimized_Access := 'TRUE' }
AUTHOR : Simatic
FAMILY : IEC
NAME : IEC_TMR
VERSION : 1.0
// stored: InstanceOfName IEC_TIMER
"IEC_TIMER"
BEGIN
END_DATA_BLOCK

DATA_BLOCK "IEC_Counter_0_DB_3"   // DB15
{ S7_Optimized_Access := 'TRUE' }
AUTHOR : SIMATIC
FAMILY : IEC
NAME : DCNTR
VERSION : 1.2
// stored: InstanceOfName IEC_DCOUNTER
"IEC_DCOUNTER"
BEGIN
END_DATA_BLOCK

DATA_BLOCK "IEC_Timer_0_DB_4"   // DB16
{ S7_Optimized_Access := 'TRUE' }
AUTHOR : Simatic
FAMILY : IEC
NAME : IEC_TMR
VERSION : 1.0
// stored: InstanceOfName IEC_TIMER
"IEC_TIMER"
BEGIN
END_DATA_BLOCK

DATA_BLOCK "IEC_Timer_0_DB_5"   // DB17
{ S7_Optimized_Access := 'TRUE' }
AUTHOR : Simatic
FAMILY : IEC
NAME : IEC_TMR
VERSION : 1.0
// stored: InstanceOfName IEC_TIMER
"IEC_TIMER"
BEGIN
END_DATA_BLOCK

DATA_BLOCK "IEC_Timer_0_DB_7"   // DB21
{ S7_Optimized_Access := 'TRUE' }
AUTHOR : Simatic
FAMILY : IEC
NAME : IEC_TMR
VERSION : 1.0
// stored: InstanceOfName IEC_TIMER
"IEC_TIMER"
BEGIN
END_DATA_BLOCK

DATA_BLOCK "IEC_Timer_0_DB_13"   // DB22
{ S7_Optimized_Access := 'TRUE' }
AUTHOR : Simatic
FAMILY : IEC
NAME : IEC_TMR
VERSION : 1.0
// stored: InstanceOfName IEC_TIMER
"IEC_TIMER"
BEGIN
END_DATA_BLOCK

DATA_BLOCK "IEC_Timer_0_DB_14"   // DB23
{ S7_Optimized_Access := 'TRUE' }
AUTHOR : Simatic
FAMILY : IEC
NAME : IEC_TMR
VERSION : 1.0
// stored: InstanceOfName IEC_TIMER
"IEC_TIMER"
BEGIN
END_DATA_BLOCK

DATA_BLOCK "IEC_Timer_0_DB_15"   // DB24
{ S7_Optimized_Access := 'TRUE' }
AUTHOR : Simatic
FAMILY : IEC
NAME : IEC_TMR
VERSION : 1.0
// stored: InstanceOfName IEC_TIMER
"IEC_TIMER"
BEGIN
END_DATA_BLOCK

DATA_BLOCK "IEC_Timer_0_DB_16"   // DB25
{ S7_Optimized_Access := 'TRUE' }
AUTHOR : Simatic
FAMILY : IEC
NAME : IEC_TMR
VERSION : 1.0
// stored: InstanceOfName IEC_TIMER
"IEC_TIMER"
BEGIN
END_DATA_BLOCK

DATA_BLOCK "IEC_Timer_0_DB_17"   // DB26
{ S7_Optimized_Access := 'TRUE' }
AUTHOR : Simatic
FAMILY : IEC
NAME : IEC_TMR
VERSION : 1.0
// stored: InstanceOfName IEC_TIMER
"IEC_TIMER"
BEGIN
END_DATA_BLOCK

DATA_BLOCK "IEC_Timer_0_DB_18"   // DB27
{ S7_Optimized_Access := 'TRUE' }
AUTHOR : Simatic
FAMILY : IEC
NAME : IEC_TMR
VERSION : 1.0
// stored: InstanceOfName IEC_TIMER
"IEC_TIMER"
BEGIN
END_DATA_BLOCK

DATA_BLOCK "IEC_Timer_0_DB_19"   // DB28
{ S7_Optimized_Access := 'TRUE' }
AUTHOR : Simatic
FAMILY : IEC
NAME : IEC_TMR
VERSION : 1.0
// stored: InstanceOfName IEC_TIMER
"IEC_TIMER"
BEGIN
END_DATA_BLOCK

DATA_BLOCK "IEC_Timer_0_DB_20"   // DB31
{ S7_Optimized_Access := 'TRUE' }
AUTHOR : Simatic
FAMILY : IEC
NAME : IEC_TMR
VERSION : 1.0
// stored: InstanceOfName IEC_TIMER
"IEC_TIMER"
BEGIN
END_DATA_BLOCK

DATA_BLOCK "IEC_Timer_0_DB_21"   // DB56
{ S7_Optimized_Access := 'TRUE' }
AUTHOR : Simatic
FAMILY : IEC
NAME : IEC_TMR
VERSION : 1.0
// stored: InstanceOfName IEC_TIMER
"IEC_TIMER"
BEGIN
END_DATA_BLOCK

DATA_BLOCK "IEC_Timer_0_DB_22"   // DB57
{ S7_Optimized_Access := 'TRUE' }
AUTHOR : Simatic
FAMILY : IEC
NAME : IEC_TMR
VERSION : 1.0
// stored: InstanceOfName IEC_TIMER
"IEC_TIMER"
BEGIN
END_DATA_BLOCK

// folder: Valve_o/c

DATA_BLOCK "Valve_o/c_fb_Arrey_DB"   // DB18
{ S7_Optimized_Access := 'TRUE' }
VERSION : 0.1
// stored: InstanceOfName Valve_o/c_fb_Arrey
"Valve_o/c_fb_Arrey"
BEGIN
END_DATA_BLOCK

DATA_BLOCK "Valve_o/c_fb_Arrey_old_DB"   // DB55
{ S7_Optimized_Access := 'TRUE' }
VERSION : 0.1
// stored: InstanceOfName Valve_o/c_fb_Arrey_old
"Valve_o/c_fb_Arrey_old"
BEGIN
END_DATA_BLOCK

// folder: _DATA-FOR_HMI

DATA_BLOCK "__MainBlock"   // DB32
{ S7_Optimized_Access := 'FALSE' }
VERSION : 0.1
   VAR
      DI : Array[0..30] of "ty_DI";
      Pump : Array[1..6] of "ty_Pump";
      AI : Array[1..12] of "ty_AI";
      "Valve_o/c" : Array[1..20] of "ty_Valve";
      Valve_Regul : Array[1..3] of "ty_Valve-regul";
      PID : Array[1..5] of Struct
         k_p : Real;
         k_I : Real;
         k_D : Real;
      END_STRUCT;
   END_VAR
BEGIN
   PID[1].k_p := 1.0;
   PID[1].k_I := 20.0;
   PID[2].k_p := 1.0;
   PID[2].k_I := 20.0;
   PID[3].k_p := 1.0;
   PID[3].k_I := 20.0;
   PID[4].k_p := 1.0;
   PID[4].k_I := 20.0;
   PID[5].k_p := 1.0;
   PID[5].k_I := 20.0;
   // AI[1] : Темп входа пива PT100
   // AI[2] : Темп выхода пива PT100
   // AI[3] : Темп ГВ - нагрев PT100
   // AI[4] : Темп Гликоль PT100
   // AI[5] : ТЕмп емкость PT100
   // AI[6] : Темп выход продукт ТТ6 4-20 мА
   // AI[7] : Расходомер 4-20
   // AI[8] : Датчик давления 4-20
   // AI[9] : Датчик давления 4-20
   // AI[10] : Датчик давления 4-20
   // AI[11] : Датчик веса буфера
   // AI[12] : Датчик концентрации
   // Valve_Regul[1] : Клапан НАГРЕВА
   // Valve_Regul[2] : Клапан Охлаждения
   // Valve_Regul[3] : Клапан Давления
END_DATA_BLOCK

// folder: _DB

DATA_BLOCK "fb_Valve-regul_DB"   // DB13
{ S7_Optimized_Access := 'TRUE' }
VERSION : 0.1
// stored: InstanceOfName fb_Valve-regul
"fb_Valve-regul"
BEGIN
END_DATA_BLOCK

DATA_BLOCK "fb_Wash_In_DB"   // DB20
{ S7_Optimized_Access := 'TRUE' }
VERSION : 0.1
// stored: InstanceOfName fb_Wash_In
"fb_Wash_In"
BEGIN
END_DATA_BLOCK

DATA_BLOCK "FB_Аварии_DB"   // DB38
{ S7_Optimized_Access := 'FALSE' }
VERSION : 0.1
// stored: InstanceOfName FB_Аварии
"FB_Аварии"
BEGIN
END_DATA_BLOCK

DATA_BLOCK "FB_Emergency_DB"   // DB39
{ S7_Optimized_Access := 'FALSE' }
VERSION : 0.1
// stored: InstanceOfName FB_Аварии
"FB_Аварии"
BEGIN
END_DATA_BLOCK

DATA_BLOCK "R_trig_All_Auto"   // DB52
{ S7_Optimized_Access := 'TRUE' }
VERSION : 0.1
// stored: InstanceOfName R_trig
"R_trig"
BEGIN
END_DATA_BLOCK

// folder: (top level)

FUNCTION_BLOCK "fb_Valve-regul"   // FB5, SCL
{ S7_Optimized_Access := 'TRUE' }
VERSION : 0.1
   VAR_IN_OUT
      aValve : Array[*] of "ty_Valve-regul";
   END_VAR
   VAR
      i : Int;
   END_VAR
   VAR_TEMP
      SizeArray : Int;
      rSetpoint : Real;
   END_VAR
BEGIN
   //Определение размера массива подаваемого на вход
   //
   #SizeArray := UPPER_BOUND(ARR := #aValve, DIM := 1);

   //ВНИМАТЕЛЬНО С МАССИВОМ ОБЯЗАТЕЛЬНО С КАКОГО НОМЕРА НАЧИНАЕТСЯ ТАКОЙ УКАЗЫВАТЬ В FOR ЕСЛИ МАССИВ С 0 ТО И FOR С 0 ЕСЛИ С 1 ТО И FOR С 1
   //
   FOR #i := 1 TO #SizeArray DO

       // =========================================
       // Выбор уставки и DO в зависимости от режима
       // =========================================
       IF #aValve[#i].bManualMode THEN
           #rSetpoint := #aValve[#i].rManualSetpoint;
           #aValve[#i].bOut_OpenClose := #aValve[#i].bManualOpenClose;
       ELSE
           #rSetpoint := #aValve[#i].rAutoSetpoint;
           #aValve[#i].bOut_OpenClose := #aValve[#i].bAutoOpenClose;
       END_IF;

       // =========================================
       // Ограничение 0…100 %
       // =========================================
       IF #rSetpoint < 0.0 THEN
           #rSetpoint := 0.0;
       ELSIF #rSetpoint > 100.0 THEN
           #rSetpoint := 100.0;
       END_IF;

       // =========================================
       // % → AO
       // =========================================
       #aValve[#i].iAnalogOutput :=
       REAL_TO_INT((#rSetpoint / 100.0) * 27648.0);

       // =========================================
       // Вывод на HMI
       // =========================================
       #aValve[#i].rValvePosPercent := #rSetpoint;

       // =========================================
       // Статус клапана
       // DO обязателен + % > 0
       // =========================================
       IF (#rSetpoint > 0.0) AND #aValve[#i].bOut_OpenClose THEN
           #aValve[#i].bStatusValveOpen := TRUE;
       ELSE
           #aValve[#i].bStatusValveOpen := FALSE;
       END_IF;

   END_FOR;
END_FUNCTION_BLOCK

FUNCTION_BLOCK "fb_Wash_In"   // FB6, SCL
{ S7_Optimized_Access := 'TRUE' }
VERSION : 0.1
   VAR_INPUT
      bCmdWashStart : Bool;   // импульс "Пуск мойки"
      bCmdWashStop : Bool;   // // импульс "Стоп мойки"
      bSelAlkali : Bool;   // выбрана щелочная мойка
      bSelAcid : Bool;   // выбрана кислотная мойка
      bZS2_PosOK : Bool;   // датчик положения "калача"
      bLevelLS1 : Bool;   // нижний уровень емкости
      bFlowPresent : Bool;   // есть поток
      bWaterPulse : Bool;   // импульс счетчика воды
      rConcActual : Real;   // текущая концентрация
      rTempActual : Real;   // текущая температура
      rTenpDelta : Real;   // Дельта температуры
      bAlarm : Bool;   // общая авария
   END_VAR
   VAR_OUTPUT
      bWashActive : Bool;
      iStep : Int;   // текущий шаг мойки
      iWaterCounter : Int;
      tTimeProcess : DInt;   // Пройденное время в сек
      rTempSet_Out : Real;   // уставка температуры
      bWashValve1 : Bool;
      bWashValve2 : Bool;
      bWashValve4 : Bool;
      bWashValve5 : Bool;
      bWashValve6 : Bool;
      bWashValve7 : Bool;
      bWashValve8 : Bool;
      bWashValve9 : Bool;
      bWashValve10 : Bool;
      bWashValve11 : Bool;
      bWashValve12 : Bool;
      bWashValve13 : Bool;
      bWashValve14 : Bool;
      bWashValve16 : Bool;
      bWashPump1 : Bool;
      bWashPump2 : Bool;
      bWashPump3 : Bool;
      bWashPump4 : Bool;
      bWashPump5 : Bool;
      bWashPump15 : Bool;
      bWashPump17 : Bool;
   END_VAR
   VAR
      iNextStep : Int;
      rStartPuls : "R_trig";   // Импульс по сигналу R_trig_Out
      rStopPuls : "R_trig";   // Импульс по сигналу R_trig_Out
      rWaterTrig : "R_trig";   // Импульс для счетчика
      rtrig_NextStep : "R_trig";
      tStepTimer : TONR_TIME;   // универсальный таймер шага
      tFlipTimer : TON_TIME;   // таймер флипования
      tChemPulse : TON_TIME;   // импульс подачи химии
      tChemPause : TON_TIME;   // пауза между импульсами
      TON_Flip : TON_TIME;   // Время перехода для флипования
      TON_FlipPause : TON_TIME;
      bFlipState : Bool;   // true = 4 valve - Open
      bConcOK : Bool;
      bTempOK : Bool;
      bTemp_Ok : Bool;   // Температура готова
      bConcentrat_Ok : Bool;   // Концентрат готов
      bFlip_En : Bool;   // Включение флипования
      iflip_step : Int;   // Шаг для флипования
   END_VAR
BEGIN

   REGION NextStep_for test

       #rtrig_NextStep(In := "nextStep");
       IF #rtrig_NextStep.Q THEN
           #iStep := #iStep + 10;
       END_IF;

   END_REGION


   REGION _R_Trig
       // --- Триггеры ---

       #rStartPuls(In := #bCmdWashStart);
       #rStopPuls(In := #bCmdWashStop);
       #rWaterTrig(In := #bWaterPulse);


   END_REGION

   REGION Alarm

       // --- Авария или стоп ---
       IF #bAlarm OR #rStopPuls.Q THEN
           #iStep := 0;
       END_IF;

   END_REGION

   REGION Время для дисплея
       // Время процесса

       #tTimeProcess := #tStepTimer.ET; //Время в мссекундах

   END_REGION


   REGION Инициализация закрытых клапанов
       // Клапана и насосы в off

       //Закрываем клапана
       #bWashValve1 := #bWashValve2 := #bWashValve4 := #bWashValve5 := #bWashValve6 := #bWashValve7 := #bWashValve8 :=
       #bWashValve9 := #bWashValve10 := #bWashValve11 := #bWashValve12 := #bWashValve13 := #bWashValve14 :=
       #bWashValve16 := FALSE;
       //Стоп насосы

       #bWashPump1 := #bWashPump2 := #bWashPump3 := #bWashPump4 := #bWashPump5 := #bWashPump15 := #bWashPump17 := FALSE;
   END_REGION

   REGION Наведение концентрации
       // Наводим растовр - задаем время импульса и паузу между импульсами

       IF (#iStep = 50 OR #iStep = 60 OR #iStep = 110 OR #iStep = 120) THEN

           #tChemPulse(IN := NOT #bConcentrat_Ok AND NOT #tChemPause.Q,
                           PT := "Уставки_Мойка_Вн".dwПаузыИмпНаведения * 1000);

               #tChemPause(IN := #tChemPulse.Q,
                           PT := "Уставки_Мойка_Вн".dwВремяИмпНаведения * 1000);
           END_IF;
   END_REGION

   REGION Флипование
       // Флипование если переменна #bFlip_En = true
       // 
       IF #bFlip_En THEN
           CASE #iflip_step OF

               0:
                   //Стоп флип
                   #bWashValve4 := FALSE;
                   #bWashValve5 := FALSE;
                   #bWashValve7 := FALSE;
                   #bWashValve8 := FALSE;
                   #TON_Flip(IN := FALSE,
                             PT := t#0s);
                   #TON_FlipPause(IN := FALSE,
                                  PT := t#0s);
                   #iflip_step := 1;

               1:  //Флип клапан 4

                   #TON_Flip.TON(IN := true, PT := "Уставки_Мойка_Вн"."dwВремяФлипованияКл,сек" * 1000);   //Time for next step

                   #bWashValve4 := TRUE;
                   #bWashValve5 := FALSE;
                   #bWashValve7 := FALSE;
                   #bWashValve8 := FALSE;

                           //Переход на следующий шаг по завершению таймера
                   IF #TON_Flip.Q THEN
                               #iflip_step := 2;
                               #TON_Flip.TON(IN := FALSE, PT := "Уставки_Мойка_Вн"."dwВремяФлипованияКл,сек" * 1000);
                   END_IF;

               2:  //Флип клапан 8
                   #TON_Flip.TON(IN := true, PT := "Уставки_Мойка_Вн"."dwВремяФлипованияКл,сек" * 1000);   //Time for next step

                   #bWashValve4 := FALSE;
                   #bWashValve5 := FALSE;
                   #bWashValve7 := TRUE;
                   #bWashValve8 := TRUE;

                   IF #TON_Flip.Q THEN
                               #iflip_step := 3;
                               #TON_Flip.TON(IN := FALSE,PT := "Уставки_Мойка_Вн"."dwВремяФлипованияКл,сек" * 1000);
                   END_IF;

               3: //Флип клапан 8

                   #TON_Flip.TON(IN := true, PT := "Уставки_Мойка_Вн"."dwВремяФлипованияКл,сек" * 1000);   //Time for next step
                   #bWashValve4 := FALSE;
                   #bWashValve5 := FALSE;
                   #bWashValve7 := TRUE;
                   #bWashValve8 := TRUE;

                   IF #TON_Flip.Q THEN

                       #bWashValve4 := FALSE;
                       #bWashValve5 := FALSE;
                       #bWashValve7 := TRUE;
                       #bWashValve8 := FALSE;


                       #TON_FlipPause.TON(IN := TRUE, PT := "Уставки_Мойка_Вн"."dwВремяПаузыФлипованияКл,сек_1" * 1000);
                   END_IF;

                   IF #TON_FlipPause.Q THEN
                       #iflip_step := 0;
                       #TON_FlipPause(IN := FALSE,
                                      PT := t#0s);
                   END_IF;



           END_CASE;

       ELSE
           #bWashValve4 := FALSE;
           #bWashValve7 := FALSE;
           #bWashValve8 := FALSE;
           #iflip_step := 0;
       END_IF;
       //....Сброс переменной.....
       #bFlip_En := FALSE;
   END_REGION


   // --- Старт мойки ---
   IF #rStartPuls.Q AND NOT #bWashActive THEN
       #bWashActive := TRUE;
       #iStep := 10;
       #iWaterCounter := 0;
       #tStepTimer(IN := false, PT := t#0s, R := TRUE);
   END_IF;


   IF #bWashActive THEN

       CASE #iStep OF

               // --------------------------------------------------
           0:  // ожидание
               // --------------------------------------------------

               //Закрываем клапана
               #bWashValve1 := #bWashValve2 := #bWashValve4 := #bWashValve5 := #bWashValve6 := #bWashValve7 := #bWashValve8 :=
               #bWashValve9 := #bWashValve10 := #bWashValve11 := #bWashValve12 := #bWashValve13 := #bWashValve14 := 
               #bWashValve16 := FALSE;
               //Стоп насосы

               #bWashPump1 := #bWashPump2 := #bWashPump3 := #bWashPump4 := #bWashPump5 := #bWashPump15 := #bWashPump17 := FALSE;

               //Ожидание Старта
               #bWashActive := FALSE;

               // --------------------------------------------------
           10: // Наполнение водой по счетчику
               // --------------------------------------------------
               #bWashValve1 := TRUE;   // вход воды
               #bWashValve7 := TRUE;
               #bWashValve8 := FALSE;
               #bWashValve13 := TRUE;

               #bWashPump1 := TRUE;
               #bWashPump2 := TRUE;

               //Подсчет кол-ва литров 
               IF #rWaterTrig.Q THEN
                   #iWaterCounter := #iWaterCounter + 1;
               END_IF;

               // Условие окончания наполнения
               IF #iWaterCounter >= "Уставки_Мойка_Вн".iCount_Water_Наполнение THEN   // Наполнение водой по счтчику
                   #iWaterCounter := 0;
                   #iStep := 20;
               END_IF;


               // --------------------------------------------------
           20: // Циркуляция воды
               // --------------------------------------------------
               // обязательное условие
               IF NOT #bZS2_PosOK THEN
                                   // ждем правильного положения
                                   // Закрыть все клпана и стоп насосы
                   #tStepTimer(IN := FALSE,PT:= t#0s, R := FALSE);


               ELSE
                   #bWashValve2 := TRUE;
                   #bWashValve6 := TRUE;
                   #bWashValve9 := TRUE;
                   #bWashValve11 := TRUE;
                   #bWashValve13 := TRUE;

                   #bWashPump1 := TRUE;
                   #bWashPump2 := TRUE;
                   #bWashPump3 := TRUE;
                   #bWashPump4 := TRUE;

                   #rTempSet_Out := "Уставки_Мойка_Вн".rSet_Temp_Nagrev_Вода;

                   // --- Флипование клапанов 4 и 7 и 8 ---
                   // 

                   #bFlip_En := TRUE;


                   // Таймер циркуляции
                   #tStepTimer(IN := TRUE,
                               PT := "Уставки_Мойка_Вн"."dwВремяЦиркуляции,мин"*60000, R := FALSE); //  уставка 
                   IF #tStepTimer.Q THEN
                       #tStepTimer (IN := FALSE, PT := t#0s, R:= TRUE);
                       #iStep := 30;
                   END_IF;
               END_IF;


               // --------------------------------------------------
           30: // Слив воды
               // --------------------------------------------------
               #bWashValve2 := TRUE;
               #bWashValve5 := TRUE;   // дренаж (НО)
               #bWashValve6 := TRUE;
               #bWashValve9 := TRUE;

               #bWashPump1 := TRUE;
               #bWashPump2 := TRUE;
               #bWashPump3 := TRUE;

               IF NOT #bLevelLS1 OR NOT #bFlowPresent THEN
                   // выбор следующего шага
                   IF #bSelAlkali THEN
                       #iStep := 40; // щелочная мойка
                   ELSIF #bSelAcid THEN
                       #iStep := 100; // кислотная мойка
                   ELSE
                       #iStep := 0;
                   END_IF;
               END_IF;

               // --------------------------------------------------
           40: // Наполнение щелочной мойки
               // --------------------------------------------------
               #bWashValve1 := TRUE;
               #bWashValve7 := TRUE;
               #bWashValve8 := TRUE;
               #bWashValve13 := TRUE;

               #bWashPump1 := TRUE;
               #bWashPump2 := TRUE;

               IF #rWaterTrig.Q THEN
                   #iWaterCounter := #iWaterCounter + 1;
               END_IF;

               IF #iWaterCounter >= "Уставки_Мойка_Вн".iCount_Water_Наполнение THEN   //Уставка такая же как и в наполнении при ополаскивании
                   #iWaterCounter := 0;
                   #iStep := 50;
               END_IF;

               // --------------------------------------------------
           50: // Наведение концентрации и температуры (щелочь)
               // --------------------------------------------------
               #bWashValve2 := TRUE;
               #bWashValve6 := TRUE;
               #bWashValve7 := TRUE;
               #bWashValve9 := TRUE;
               #bWashValve11 := TRUE;  //Нагрев
               #bWashValve13 := TRUE;

               //---------Концентрат----------
               #bWashValve14   := #tChemPulse.Q;
               #bWashPump15    := #tChemPulse.Q;

               #bWashPump1 := TRUE;
               #bWashPump2 := TRUE;
               #bWashPump3 := TRUE;
               #bWashPump4 := TRUE;

               // --- Флипование клапанов 4 и 7 и 8 ---
               // 
                      // #bFlip_En := TRUE;

               // --- Контроль температуры ---

               #bTemp_Ok := (#rTempActual >= "Уставки_Мойка_Вн".rSet_Temp_Nagrev_Щелочь - #rTenpDelta);

               #rTempSet_Out := "Уставки_Мойка_Вн".rSet_Temp_Nagrev_Щелочь;
               // --- Контроль Концентрации ---

               #bConcentrat_Ok := #rConcActual > ("Уставки_Мойка_Вн".rSet_Concentr_Щелочь - "Уставки_Мойка_Вн".rSet_Conc_Delta);

              (* IF NOT #bConcentrat_Ok THEN

                   #tChemPulse(IN := NOT #bConcentrat_Ok AND NOT #tChemPulse.Q,
                               PT := "Уставки_Мойка_Вн".dwПаузыИмпНаведения * 1000);

                   #tChemPause(IN := #tChemPause.Q,
                               PT := "Уставки_Мойка_Вн".dwВремяИмпНаведения*1000);
               END_IF;
               *)

               IF #bTemp_Ok AND #bConcentrat_Ok THEN
                   #iStep := 60;
               END_IF;


               // --------------------------------------------------
           60: // Циркуляция щелочи
               // --------------------------------------------------
               // 
               // обязательное условие
               IF NOT #bZS2_PosOK THEN
                   // ждем правильного положения
                   // Закрыть все клпана и стоп насосы
                   #tStepTimer(IN := FALSE,
                               PT := t#0s,
                               R := FALSE);


               ELSE
                   #bWashValve2 := TRUE;
                   #bWashValve6 := TRUE;
                   #bWashValve9 := TRUE;
                   #bWashValve13 := TRUE;

                   #bWashPump1 := TRUE;
                   #bWashPump2 := TRUE;
                   #bWashPump3 := TRUE;
                   #bWashPump4 := TRUE;

                   #bWashValve11 := TRUE;

                   //---------Концентрат----------
                   #bWashValve14 := #tChemPulse.Q;
                   #bWashPump15 := #tChemPulse.Q;

                   // --- Флипование клапанов 4 и 7 и 8 ---
                   // 
                        #bFlip_En := TRUE;

                   // --- Поддержка концентрации ---
                   // 
                        #bConcentrat_Ok := #rConcActual > ("Уставки_Мойка_Вн".rSet_Concentr_Щелочь - "Уставки_Мойка_Вн".rSet_Conc_Delta);
                        #bTemp_Ok := (#rTempActual >= "Уставки_Мойка_Вн".rSet_Temp_Nagrev_Щелочь - #rTenpDelta);

             (*      IF NOT #bConcentrat_Ok THEN

                       #tChemPulse(IN := NOT #bConcentrat_Ok AND NOT #tChemPulse.Q,
                                   PT := "Уставки_Мойка_Вн".dwПаузыИмпНаведения * 1000);

                       #tChemPause(IN := #tChemPause.Q,
                                   PT := "Уставки_Мойка_Вн".dwВремяИмпНаведения * 1000);
                   END_IF;
                *)   


                   // -------Время циркуляции щелочи------
                        #tStepTimer(IN := #bConcentrat_Ok AND #bTemp_Ok,
                               PT := "Уставки_Мойка_Вн"."dwВремяЩОЛОЧЬ_Циркул,ми" * 60000,
                               R := FALSE);

                   IF #tStepTimer.Q THEN

                       #tStepTimer(IN := FALSE,
                                   PT := t#0s,
                                   R := TRUE);
                       #iStep := 70;
                   END_IF;
               END_IF;

               // --------------------------------------------------
           70: // Слив щелочи
               // --------------------------------------------------
               #bWashValve2 := TRUE;
               #bWashValve5 := TRUE;
               #bWashValve6 := TRUE;
               #bWashValve9 := TRUE;
               #bWashValve13 := TRUE;

               #bWashPump1 := TRUE;
               #bWashPump2 := TRUE;
               #bWashPump3 := TRUE;

               IF NOT #bLevelLS1 OR NOT #bFlowPresent THEN
                   #iStep := 80;
               END_IF;

               // --------------------------------------------------
           80: // Полоскание после щелочи
               // --------------------------------------------------
               #bWashValve1 := TRUE;
               #bWashValve7 := TRUE;
               #bWashValve8 := TRUE;
               #bWashValve13 := TRUE;

               #bWashPump1 := TRUE;
               #bWashPump2 := TRUE;

               IF #rWaterTrig.Q THEN
                   #iWaterCounter := #iWaterCounter + 1;
               END_IF;

                   ///------------ Контроль счетчика для ополаскивания или уровень конценрации щелочи в вода----------------
                   //
               IF (#iWaterCounter >= "Уставки_Мойка_Вн".iCount_Water_ПолосЩелочи)OR
                  (#rConcActual <= "Уставки_Мойка_Вн".rSet_Concentr_Вода)
               THEN
                   #iWaterCounter := 0;
                   #iStep := 90;
               END_IF;

               // --------------------------------------------------
           90: // Слив после щелочи
               // --------------------------------------------------
               #bWashValve2 := TRUE;
               #bWashValve5 := TRUE;
               #bWashValve6 := TRUE;
               #bWashValve9 := TRUE;

               #bWashPump1 := TRUE;
               #bWashPump2 := TRUE;
               #bWashPump3 := TRUE;

               IF NOT #bLevelLS1 OR NOT #bFlowPresent THEN
                   IF #bSelAcid THEN
                       #iStep := 100;   // переход к кислоте
                   ELSE
                       #iStep := 170;
                   END_IF;
               END_IF;

               // --------------------------------------------------
           100: // Наполнение Кислотной мойки
               // --------------------------------------------------
               #bWashValve1 := TRUE;
               #bWashValve7 := TRUE;
               #bWashValve8 := TRUE;
               #bWashValve13 := TRUE;

               #bWashPump1 := TRUE;
               #bWashPump2 := TRUE;

               IF #rWaterTrig.Q THEN
                   #iWaterCounter := #iWaterCounter + 1;
               END_IF;

               IF #iWaterCounter >= "Уставки_Мойка_Вн".iCount_Water_Наполнение THEN   //Уставка такая же как и в наполнении при ополаскивании
                   #iWaterCounter := 0;
                   #iStep := 110;
               END_IF;

               // --------------------------------------------------
           110: // Наведение концентрации и температуры (Кислота)
               // --------------------------------------------------
               #bWashValve2 := TRUE;
               #bWashValve6 := TRUE;
               #bWashValve7 := TRUE;
               #bWashValve9 := TRUE;
               #bWashValve11 := TRUE;  //Нагрев
               #bWashValve13 := TRUE;

               //---------Концентрат----------
               #bWashValve16 := #tChemPulse.Q;
               #bWashPump17 := #tChemPulse.Q;

               #bWashPump1 := TRUE;
               #bWashPump2 := TRUE;
               #bWashPump3 := TRUE;
               #bWashPump4 := TRUE;


               // --- Флипование клапанов 4 и 7 и 8 ---
               // 
                      //  #bFlip_En := TRUE;

               // --- Контроль температуры ---

               #bTemp_Ok := (#rTempActual >= "Уставки_Мойка_Вн".rSet_Temp_Nagrev_Кислота - #rTenpDelta);

               #rTempSet_Out := "Уставки_Мойка_Вн".rSet_Temp_Nagrev_Кислота;

               // --- Контроль Концентрации ---

               #bConcentrat_Ok := #rConcActual > ("Уставки_Мойка_Вн".rSet_Concentr_Кислота - "Уставки_Мойка_Вн".rSet_Conc_Delta);

        (*       IF NOT #bConcentrat_Ok THEN

                   #tChemPulse(IN := NOT #bConcentrat_Ok AND NOT #tChemPulse.Q,
                               PT := "Уставки_Мойка_Вн".dwПаузыИмпНаведения * 1000);

                   #tChemPause(IN := #tChemPause.Q,
                               PT := "Уставки_Мойка_Вн".dwВремяИмпНаведения * 1000);
               END_IF;
         *)      
         //Переход на следующий шаг
         //
               IF #bTemp_Ok AND #bConcentrat_Ok THEN
                   #iStep := 120;
               END_IF;


               // --------------------------------------------------
           120: // Циркуляция кислоты
               // --------------------------------------------------
               // 
               // обязательное условие
               IF NOT #bZS2_PosOK THEN
                   // ждем правильного положения
                   // Закрыть все клпана и стоп насосы
                   #tStepTimer(IN := FALSE,
                               PT := t#0s,
                               R := FALSE);


               ELSE
                   #bWashValve2 := TRUE;
                   #bWashValve6 := TRUE;
                   #bWashValve7 := TRUE;
                   #bWashValve9 := TRUE;
                   #bWashValve13 := TRUE;

                   #bWashPump1 := TRUE;
                   #bWashPump2 := TRUE;
                   #bWashPump3 := TRUE;
                   #bWashPump4 := TRUE;

                   #bWashValve11 := TRUE;

                   #bWashValve16 := #tChemPulse.Q;
                   #bWashPump17 := #tChemPulse.Q;


                   // --- Флипование клапанов 4 и 7 и 8 ---
                   // 
                           #bFlip_En := TRUE;

                   // --- Поддержка концентрации ---
                   // 
                           #bConcentrat_Ok := #rConcActual > ("Уставки_Мойка_Вн".rSet_Concentr_Кислота - "Уставки_Мойка_Вн".rSet_Conc_Delta);

                           #bTemp_Ok := (#rTempActual >= "Уставки_Мойка_Вн".rSet_Temp_Nagrev_Кислота - #rTenpDelta);

                (*   IF NOT #bConcentrat_Ok THEN

                       #tChemPulse(IN := NOT #bConcentrat_Ok AND NOT #tChemPulse.Q,
                                   PT := "Уставки_Мойка_Вн".dwПаузыИмпНаведения * 1000);

                       #tChemPause(IN := #tChemPause.Q,
                                   PT := "Уставки_Мойка_Вн".dwВремяИмпНаведения * 1000);
                   END_IF;
               *)    
                           #tStepTimer(IN := #bConcentrat_Ok AND #bTemp_Ok,
                               PT := "Уставки_Мойка_Вн"."dwВремяЩОЛОЧЬ_Циркул,ми" * 60000,
                               R := FALSE);

                   IF #tStepTimer.Q THEN

                       #tStepTimer(IN := FALSE,
                                   PT := t#0s,
                                   R := TRUE);
                       #iStep := 130;
                   END_IF;
               END_IF;

               // --------------------------------------------------
           130: // Слив Кислоты
               // --------------------------------------------------
               #bWashValve2 := TRUE;
               #bWashValve5 := TRUE;
               #bWashValve6 := TRUE;
               #bWashValve9 := TRUE;
               #bWashValve13 := TRUE;

               #bWashPump1 := TRUE;
               #bWashPump2 := TRUE;
               #bWashPump3 := TRUE;

               IF NOT #bLevelLS1 OR NOT #bFlowPresent THEN
                   #iStep := 140;
               END_IF;

               // --------------------------------------------------
           140: // Полоскание после К
               // --------------------------------------------------
               #bWashValve1 := TRUE;
               #bWashValve7 := TRUE;
               #bWashValve8 := TRUE;
               #bWashValve13 := TRUE;

               #bWashPump1 := TRUE;
               #bWashPump2 := TRUE;

               IF #rWaterTrig.Q THEN
                   #iWaterCounter := #iWaterCounter + 1;
               END_IF;

               ///------------ Контроль счетчика для ополаскивания или уровень конценрации щелочи в вода----------------
               //
               IF (#iWaterCounter >= "Уставки_Мойка_Вн".iCount_Water_ПолосКислоты) OR
                   (#rConcActual <= "Уставки_Мойка_Вн".rSet_Concentr_Вода)
               THEN
                   #iWaterCounter := 0;
                   #iStep := 150;
               END_IF;

               // --------------------------------------------------
           150: // Слив после Кислоты
               // --------------------------------------------------
               #bWashValve2 := TRUE;
               #bWashValve5 := TRUE;
               #bWashValve6 := TRUE;
               #bWashValve9 := TRUE;

               #bWashPump1 := TRUE;
               #bWashPump2 := TRUE;
               #bWashPump3 := TRUE;

               IF NOT #bLevelLS1 OR NOT #bFlowPresent THEN
                   #iStep := 170;
                   END_IF;




                   // --------------------------------------------------
               170: // Наполнение водой по счетчику
                   // --------------------------------------------------
                   #bWashValve1 := TRUE;   // вход воды
                   #bWashValve7 := TRUE;
                   #bWashValve8 := TRUE;
                   #bWashValve13 := TRUE;

                   #bWashPump1 := TRUE;
                   #bWashPump2 := TRUE;

                   //Подсчет кол-ва литров 
                   IF #rWaterTrig.Q THEN
                       #iWaterCounter := #iWaterCounter + 1;
                   END_IF;

                   // Условие окончания наполнения
                   IF #iWaterCounter >= "Уставки_Мойка_Вн".iCount_Water_Наполнение THEN   // Наполнение водой по счтчику
                       #iWaterCounter := 0;
                       #iStep := 180;
                   END_IF;


                   // --------------------------------------------------
               180: // Циркуляция воды
                   // --------------------------------------------------
                   // обязательное условие
                   IF NOT #bZS2_PosOK THEN
                       // ждем правильного положения
                       // Закрыть все клпана и стоп насосы
                       #tStepTimer(IN := FALSE,
                                   PT := t#0s,
                                   R := FALSE);


                   ELSE
                       #bWashValve2 := TRUE;
                       #bWashValve6 := TRUE;
                       #bWashValve7 := TRUE;
                       #bWashValve9 := TRUE;
                       #bWashValve11 := TRUE;
                       #bWashValve13 := TRUE;

                       #bWashPump1 := TRUE;
                       #bWashPump2 := TRUE;
                       #bWashPump3 := TRUE;
                       #bWashPump4 := TRUE;

                       #rTempSet_Out := "Уставки_Мойка_Вн".rSet_Temp_Nagrev_Вода;

                       // --- Флипование клапанов 4 и 7 и 8 ---
                       // 
                       #bFlip_En := TRUE;

                       // Таймер циркуляции
                       #tStepTimer(IN := TRUE,
                                   PT := "Уставки_Мойка_Вн"."dwВремяЦиркуляции,мин" * 60000,
                                   R := FALSE); //  уставка 
                       IF #tStepTimer.Q THEN
                           #tStepTimer(IN := FALSE,
                                       PT := t#0s,
                                       R := TRUE);
                           #iStep := 190;
                       END_IF;
                   END_IF;


                   // --------------------------------------------------
              190: // Слив воды
                   // --------------------------------------------------
                   #bWashValve2 := TRUE;
                   #bWashValve5 := TRUE;   // дренаж (НО)
                   #bWashValve6 := TRUE;
                   #bWashValve9 := TRUE;

                   #bWashPump1 := TRUE;
                   #bWashPump2 := TRUE;
                   #bWashPump3 := TRUE;

                   IF NOT #bLevelLS1 OR NOT #bFlowPresent THEN
                       #iStep := 0;
                   END_IF;

       END_CASE;

   END_IF;
END_FUNCTION_BLOCK

FUNCTION_BLOCK "FB_Аварии"   // FB7, SCL
{ S7_Optimized_Access := 'FALSE' }
VERSION : 0.1
   VAR_INPUT
      Rtrig_Reset : Bool;
   END_VAR
   VAR_OUTPUT
      ALARM_Active : Bool;   // Флаг активной аварии
   END_VAR
   VAR
      LatchedEmergency : Bool;   // Зафиксированная аварийная ситуация
      bAlarmAvtomats : Bool;   // Авария автоматов
      bAlarmAI : Bool;   // Авария аналоговых датчиков
      bAlarmPumps : Bool;   // Авария насосов
      bAlarmConveyors : Bool;   // Авария Конвейеров
      bAlarmFVs : Bool;   // Авария клапанов
      bAlarmDI_all : Bool;   // Авария по дискретным входам "общая"
      bAlarmLowLevel : Bool;   // Авария по низкому уровню емкостей
      bAlarmProcess : Bool;   // Аварии которые возникают в результате работы
      mReset : Bool;
      TON_LowLevel : TON_TIME;   // Таймер для аварийного уровня емкостей
      bResetaALARM : Bool;   // Сброс аварии (кнопка на панели/системе)
   END_VAR
   VAR_TEMP
      nAi : Int;
      nPump : Int;
      nConv : Int;
      nFV : Int;
      nAvtomat : Int;
      numPump : Int;
   END_VAR
BEGIN
   REGION Предварительное отрицание
       // Сброс в 0 при отсутсвии аварий для цикла и массивов
       #bAlarmAvtomats := FALSE;
       #bAlarmAI := FALSE;
       #bAlarmPumps := FALSE;
       #bAlarmConveyors := FALSE;
       #bAlarmFVs := FALSE;


   END_REGION



   //Авария автоматические выключатели
   //--------------------------
   (*
   "Alarms".Avtomat_Off[1].ALARM := NOT "Conveyor".Conveyor_1.bIn_AutomatState;
   "Alarms".Avtomat_Off[2].ALARM := NOT "Conveyor".Conveyor_2.bIn_AutomatState;
   "Alarms".Avtomat_Off[3].ALARM := NOT "Conveyor".Conveyor_3.bIn_AutomatState;
   "Alarms".Avtomat_Off[4].ALARM  :=  NOT "Pumps_1".Pump_1.bIn_AutomatState;
   "Alarms".Avtomat_Off[5].ALARM  :=  NOT "Pumps_1".Pump_2.bIn_AutomatState;
   "Alarms".Avtomat_Off[6].ALARM  :=  NOT "Pumps_1".Pump_3.bIn_AutomatState;
   "Alarms".Avtomat_Off[7].ALARM  :=  NOT "Pumps_1".Pump_4.bIn_AutomatState;
   "Alarms".Avtomat_Off[8].ALARM  :=  NOT "Pumps_1".Pump_5.bIn_AutomatState;
   "Alarms".Avtomat_Off[9].ALARM  :=  NOT "Pumps_1".Pump_6.bIn_AutomatState;
   "Alarms".Avtomat_Off[10].ALARM  :=  NOT "Pumps_1".Pump_7.bIn_AutomatState;
   "Alarms".Avtomat_Off[11].ALARM  :=  NOT "Vent".Vent_1.bIn_AutomatState;


   FOR #nAvtomat := 1 TO 11 DO
       IF "Alarms".Avtomat_Off[#nAvtomat].ALARM THEN
           #bAlarmAvtomats := TRUE;
       END_IF;
       END_FOR;
       *)

   //Авария аналоговых входов
   //--------------------------
   FOR #nAi := 1 TO 12 DO
       IF "__MainBlock".AI[#nAi].bOut_Error THEN
           #bAlarmAI := TRUE;
       END_IF;
   END_FOR;

   //Авария НАСОСОВ
   //--------------------------

   FOR #nPump := 1 TO 6 DO
       IF "__MainBlock".Pump[#nPump].bALARM THEN
           #bAlarmPumps := TRUE;
           #numPump := #nPump;

       END_IF;
   END_FOR;


   //Авария КОНВЕЙЕРОВ
   //--------------------------
   (*
   FOR #nConv := 1 TO 4 DO
       IF "Alarms".Conveyor_Alarm[#nConv].ALARM THEN
           #bAlarmConveyors := TRUE;
       END_IF;
   END_FOR;
   *)

   //Авария Клапанов
   //--------------------------

   FOR #nFV := 1 TO 20 DO
       IF "__MainBlock"."Valve_o/c"[#nFV].bValveFault THEN
           #bAlarmFVs := TRUE;
       END_IF;
   END_FOR;

   (*
   //Авария под давлению
   //--------------------------
   "AlarmPress" := "Control_Press_DB".PressWater.bAlarm_Press OR "Control_Press_DB".PressSteam.bAlarm_Press OR "Control_Press_DB".PressGlikol.bAlarm_Press;
   *)
   (*
   //Авария по нижним датчикам уровня емкостей
   //

   #bAlarmLowLevel := NOT "My_VarS".b_Woter_LowLevel_T1;
   *)

   //Авария по входам DI
   //---------------------------

   #bAlarmDI_all :=    NOT "fb_DI_Аварийный STOP" OR
                       "fb_DI_Реле давл. воздуха" OR
                       NOT "fb_DI_Реле обрыв/перекос фазы";

   //Программные Аварии - в результате процесса

                       #bAlarmProcess := "Авария давления секции пастеризации";

   //Обработка всех аварий с выводом сигнала наличия АВАРИЯ
   //----------------------------------------------------------------
                       IF #bAlarmAI OR #bAlarmPumps OR #bAlarmFVs OR #bAlarmDI_all OR #bAlarmProcess THEN

                           #ALARM_Active := TRUE;

                       END_IF;



   //Отлавливаем фронт Ресета....................................
   (*
   #bResetaALARM := #Rtrig_Reset AND NOT #mReset;
   #mReset := #Rtrig_Reset;
   *)

    //Если нужен жесткий сбро, игнорирует все аварии                      
   #bResetaALARM := #Rtrig_Reset;

   //-------------------------------------------------------------                       
                          // Сброс аварии
   IF #bResetaALARM THEN
       #ALARM_Active := FALSE;
   END_IF;
END_FUNCTION_BLOCK

FUNCTION_BLOCK "R_trig"   // FB8, SCL
{ S7_Optimized_Access := 'TRUE' }
VERSION : 0.1
   VAR_INPUT
      In : Bool;
   END_VAR
   VAR_OUTPUT
      Q : Bool;
   END_VAR
   VAR
      mIn : Bool;
   END_VAR
BEGIN
   IF #In AND NOT #mIn THEN
       #Q := TRUE;
   ELSE
       #Q := FALSE;
   END_IF;

   #mIn := #In;
END_FUNCTION_BLOCK

FUNCTION_BLOCK "Флипование"   // FB10, SCL
{ S7_Optimized_Access := 'TRUE' }
VERSION : 0.1
   VAR_INPUT
      bFlip_En : Bool;
      Time_Flip : DInt := 1;
      Time_Pause : DInt := 10;
   END_VAR
   VAR_OUTPUT
      bWashValve4 : Bool;
      bWashValve5 : Bool;
      bWashValve7 : Bool;
      bWashValve8 : Bool;
   END_VAR
   VAR
      iflip_step : Int;
      TON_Flip : TON_TIME;
      TON_Pause : TON_TIME;
      tTime_Flim_sec : DInt;
      tTime_Flim_Pause : DInt;
   END_VAR
BEGIN
   #tTime_Flim_sec := #Time_Flip * 1000;
   #tTime_Flim_Pause := #Time_Pause * 1000;

   IF #bFlip_En THEN
       CASE #iflip_step OF

           0:
               //Стоп флип
               #bWashValve4 := FALSE;
               #bWashValve5 := FALSE;
               #bWashValve7 := FALSE;
               #bWashValve8 := FALSE;
               #TON_Pause(IN := FALSE,
                          PT := t#0s);
               #iflip_step := 1;

           1:  //Флип клапан 4

               #TON_Flip.TON(IN := true,
                             PT := #tTime_Flim_sec);   //Time for next step

               #bWashValve4 := TRUE;
               #bWashValve5 := FALSE;
               #bWashValve7 := FALSE;
               #bWashValve8 := FALSE;
               #TON_Pause(IN := FALSE,
                          PT := t#0s);

               //Переход на следующий шаг по завершению таймера
               IF #TON_Flip.Q THEN
                   #iflip_step := 4;
                   #TON_Flip.TON(IN := FALSE,
                                 PT := t#0s);
               END_IF;

           2:  //Флип клапан 5 - убрал шаг пропускаю из 1 шага идем сразу в 4
               #TON_Flip.TON(IN := true,
                             PT := #tTime_Flim_sec);   //Time for next step

               #bWashValve4 := FALSE;
               #bWashValve5 := TRUE;
               #bWashValve7 := TRUE;
               #bWashValve8 := FALSE;

               //Переход на следующий шаг по завершению таймера
               IF #TON_Flip.Q THEN
                   #iflip_step := 4;
                   #TON_Flip.TON(IN := FALSE,
                                 PT := t#0s);
               END_IF;
               (*
           3: //Флип клапан 7

               #TON_Flip.TON(IN := true,
                             PT := #tTime_Flim_sec);   //Time for next step

               #bWashValve4 := FALSE;
               #bWashValve5 := FALSE;
               #bWashValve7 := TRUE;
               #bWashValve8 := FALSE;

               //Переход на следующий шаг по завершению таймера
               IF #TON_Flip.Q THEN
                   #iflip_step := 4;
                   #TON_Flip.TON(IN := FALSE,
                                 PT := t#0s);
               END_IF;
               *)
           4: //Флип клапан 8

               #TON_Flip.TON(IN := true,
                             PT := #tTime_Flim_sec);   //Time for next step

               #bWashValve4 := FALSE;
               #bWashValve5 := FALSE;
               #bWashValve7 := TRUE;
               #bWashValve8 := TRUE;

               //Переход на следующий шаг по завершению таймера
               IF #TON_Flip.Q THEN
                   #bWashValve4 := FALSE;
                   #bWashValve5 := FALSE;
                   #bWashValve7 := TRUE;
                   #bWashValve8 := FALSE;

                   #TON_Pause(IN := TRUE,
                              PT := #tTime_Flim_Pause);
               END_IF;

               IF #TON_Pause.Q THEN
                   #TON_Flip.TON(IN := FALSE,
                                 PT := t#0s);
                   #TON_Pause(IN := #TON_Flip.Q,
                              PT := t#0s);
                   #iflip_step := 1;
               END_IF;

       END_CASE;

   ELSE
       #bWashValve4 := FALSE;
       #bWashValve5 := FALSE;
       #bWashValve7 := TRUE;
       #bWashValve8 := FALSE;
       #TON_Pause(IN := FALSE,
                  PT := t#0s);
       #iflip_step := 0;
   END_IF;
   //....Сброс переменной.....
   #bFlip_En := FALSE;
END_FUNCTION_BLOCK

FUNCTION "Расчет ПЕ" : Void   // FC1, LAD
{ S7_Optimized_Access := 'FALSE' }
VERSION : 0.1
   VAR_INPUT
      "ПЕ (ед)" : Int;
      "Выдержка (сек)" : Int;
      "Производит установки (л\ч)" : Int;
      "Производит заданная (л\ч)" : Int;
   END_VAR
   VAR_OUTPUT
      "Температура пастеризации заданная (из ПЕ)" : Real;
      "Выдержка реальная_1" : Int;
   END_VAR
   VAR_TEMP
      "1" : Real;
      "выдержка реальная" : Int;
      "2" : UInt;
      "3" : Real;
      "4" : Real;
      "5" : Real;
      "6" : Real;
      "7" : Int;
      "8" : Int;
      "PE/10" : Int;
   END_VAR
BEGIN

REGION Network 1
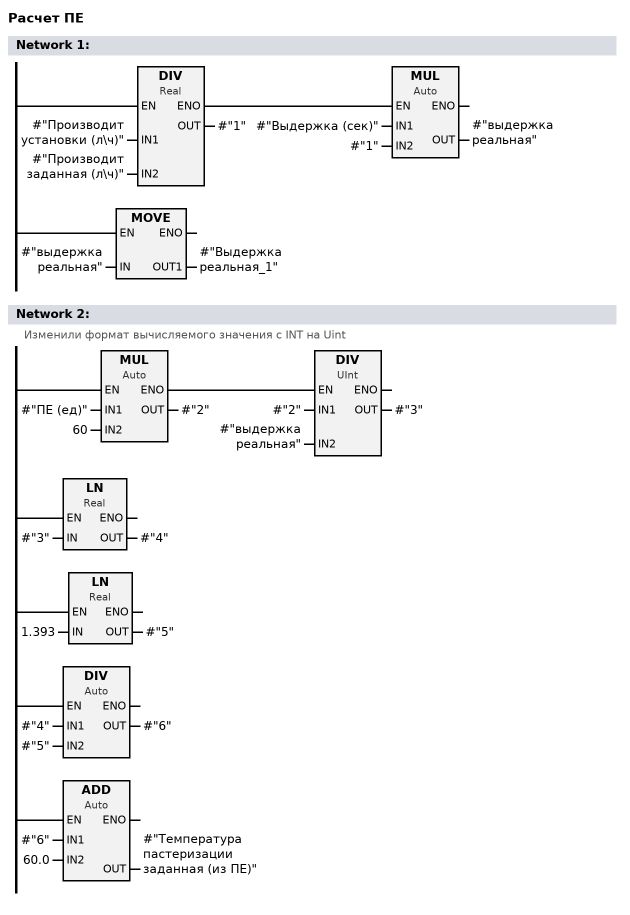
   RUNG wire#powerrail
      { S7_Templates := "SrcType := Real" } Div(in1 := #"Производит установки (л\ч)", in2 := #"Производит заданная (л\ч)", out => #"1")
      Mul(in1 := #"Выдержка (сек)", in2 := #"1", out => #"выдержка реальная")
   END_RUNG
   RUNG wire#powerrail
      Move(in := #"выдержка реальная", out1 => #"Выдержка реальная_1")
   END_RUNG
   // the same network as SCL:
   #"1" := #"Производит установки (л\ч)" / #"Производит заданная (л\ч)";
   #"выдержка реальная" := #"Выдержка (сек)" * #"1";
   #"Выдержка реальная_1" := #"выдержка реальная";
END_REGION

REGION Network 2
   // Изменили формат вычисляемого значения с INT на Uint
   #"2" := #"ПЕ (ед)" * 60;
   #"3" := #"2" / #"выдержка реальная";
   #"4" := LN(#"3");
   #"5" := LN(1.393);
   #"6" := #"4" / #"5";
   #"Температура пастеризации заданная (из ПЕ)" := #"6" + 60.0;
END_REGION
END_FUNCTION

FUNCTION "DI" : Void   // FC2, SCL
{ S7_Optimized_Access := 'TRUE' }
VERSION : 0.1
BEGIN

   REGION Присвоение входов к ФБ DI
         //Присвоение всех входов к DI.In
         //
       "__MainBlock".DI[0].In := "Аварийный STOP";
       "__MainBlock".DI[1].In := "Реле обрыв/перекос фазы";
       "__MainBlock".DI[2].In := "Работа ПЧ-1";
       "__MainBlock".DI[3].In := "Работа ПЧ-2";
       "__MainBlock".DI[4].In := "Работа ПЧ-3";
       "__MainBlock".DI[5].In := "Работа ПЧ-4";
       "__MainBlock".DI[6].In := "Работа ПЧ-5";
       "IEC_Timer_0_DB_5".TON(IN:="Реле давл. воздуха",
                              PT:=t#5s,
                              Q=>"__MainBlock".DI[7].In);

      // "__MainBlock".DI[7].In := "Реле давл. воздуха";
       "__MainBlock".DI[8].In := "Состояние V1";
       "__MainBlock".DI[9].In := "Состояние V2";
       "__MainBlock".DI[10].In := "Состояние V3";
       "__MainBlock".DI[11].In := "Состояние V4";
       "__MainBlock".DI[12].In := "Состояние V5";
       "__MainBlock".DI[13].In := "Состояние V6";
       "__MainBlock".DI[14].In := "Состояние V7";
       "__MainBlock".DI[15].In := "Состояние V8";
       "__MainBlock".DI[16].In := "Состояние V9";
       "__MainBlock".DI[17].In := "Состояние V10";
       "__MainBlock".DI[18].In := "LS1 - Низ Буфер";
       "__MainBlock".DI[19].In := "LS2 - Верх Буфер";
       "__MainBlock".DI[20].In := "LS3 - Латерн";
       "__MainBlock".DI[21].In := "Импульс с расходомера";
       "__MainBlock".DI[22].In := "Калач ZS1";
       "__MainBlock".DI[23].In := "Калач ZS2";
       "__MainBlock".DI[24].In := "Калач ZS3";
       "__MainBlock".DI[25].In := "Калач ZS4";
       "__MainBlock".DI[26].In := "Калач ZS5";
       "__MainBlock".DI[27].In := "Калач ZS6";
       "__MainBlock".DI[28].In := "Калач ZS7";





   END_REGION

   //Передача данных в блок обработки входов DI


   "DI_fb_Arrey_Old_DB"("__MainBlock".DI);

   REGION Значение выхода ФБ для программы
       //Сохранение значения обработанного входа для использования в программе
       //

       "fb_DI_Аварийный STOP" := "__MainBlock".DI[0].Out;
       "fb_DI_Реле обрыв/перекос фазы" := "__MainBlock".DI[1].Out;
       "fb_DI_Работа ПЧ-1" := "__MainBlock".DI[2].Out;
       "fb_DI_Работа ПЧ-2" := "__MainBlock".DI[3].Out;
       "fb_DI_Работа ПЧ-3" := "__MainBlock".DI[4].Out;
       "fb_DI_Работа ПЧ-4" := "__MainBlock".DI[5].Out;
       "fb_DI_Работа ПЧ-5" := "__MainBlock".DI[6].Out;
       "fb_DI_Реле давл. воздуха" := "__MainBlock".DI[7].Out;
       "fb_DI_Состояние V1" := "__MainBlock".DI[8].Out;
       "fb_DI_Состояние V2" := "__MainBlock".DI[9].Out;
       "fb_DI_Состояние V3" := "__MainBlock".DI[10].Out;
       "fb_DI_Состояние V4" := "__MainBlock".DI[11].Out;
       "fb_DI_Состояние V5" := "__MainBlock".DI[12].Out;
       "fb_DI_Состояние V6" := "__MainBlock".DI[13].Out;
       "fb_DI_Состояние V7" := "__MainBlock".DI[14].Out;
       "fb_DI_Состояние V8" := "__MainBlock".DI[15].Out;
       "fb_DI_Состояние V9" := "__MainBlock".DI[16].Out;
       "fb_DI_Состояние V10" := "__MainBlock".DI[17].Out;
       "fb_DI_LS1 - Низ Буфер" := "__MainBlock".DI[18].Out;
       "fb_DI_LS2 - Верх Буфер" := "__MainBlock".DI[19].Out;
       "fb_DI_LS3 - Латерн" := "__MainBlock".DI[20].Out;
       "fb_DI_Импульс с расходомера" := "__MainBlock".DI[21].Out;
       "fb_DI_Калач ZS1" := "__MainBlock".DI[22].Out;
       "fb_DI_Калач ZS2" := "__MainBlock".DI[23].Out;
       "fb_DI_Калач ZS3" := "__MainBlock".DI[24].Out;
       "fb_DI_Калач ZS4" := "__MainBlock".DI[25].Out;
       "fb_DI_Калач ZS5" := "__MainBlock".DI[26].Out;
       "fb_DI_Калач ZS6" := "__MainBlock".DI[27].Out;
       "fb_DI_Калач ZS7" := "__MainBlock".DI[28].Out;


   END_REGION
END_FUNCTION

FUNCTION "Pumps" : Void   // FC3, SCL
{ S7_Optimized_Access := 'TRUE' }
VERSION : 0.1
BEGIN
   //========================================== ВХОДЫ  =============================================================
   //сМОТРИ ПИД

   "__MainBlock".Pump[1].rAutoSpeed := "iPid_Out_Насос продукта-1";
   "__MainBlock".Pump[2].rAutoSpeed := "iPid_Out_Насос продукта-2";



   //

   //Насос продукта М1
   "FB_Pump_DB_1"(bManualMode := "__MainBlock".Pump[1].bManualMode,
                  bManualStart := "__MainBlock".Pump[1].bManualStart,
                  rManualSpeed := "__MainBlock".Pump[1].rManualSpeed,
                  bDryRunn := NOT "Авария низкий расход",
                  bAutoStartPerm := "__MainBlock".Pump[1].bAutoCMD,
                  rAutoSpeed := "__MainBlock".Pump[1].rAutoSpeed,
                  bАвтоматы := 1,
                  bПускатели := 1,
                  bDriveRunning := "fb_DI_Работа ПЧ-1",
                  bDriveFault := 0,
                  bResetFault := "__MainBlock".Pump[1].bResAlarm,
                  bRunCmd => "Насос М1",
                  iSpeedOut => "AO Скорость M1",
                  "rSpeedHMI(0-100)" => "__MainBlock".Pump[1]."rHMI_Speed%",
                  bPumpRunning => "__MainBlock".Pump[1].bHMI_RUN_State,
                  bPumpFault => "__MainBlock".Pump[1].bALARM,
                  iStatus => "__MainBlock".Pump[1].iHMI_Status);

   //Насос Доп продукта М2
   "FB_Pump_DB_2"(bManualMode:="__MainBlock".Pump[2].bManualMode,
                  bManualStart:="__MainBlock".Pump[2].bManualStart,
                  rManualSpeed:="__MainBlock".Pump[2].rManualSpeed,
                  bDryRunn:= NOT "Авария низкий расход",
                  bAutoStartPerm:="__MainBlock".Pump[2].bAutoCMD,
                  rAutoSpeed:="__MainBlock".Pump[2].rAutoSpeed,
                  bАвтоматы:=1,
                  bПускатели:=1,
                  bDriveRunning:="fb_DI_Работа ПЧ-2",
                  bDriveFault:=0,
                  bResetFault:="__MainBlock".Pump[2].bResAlarm,
                  bRunCmd=>"Насос М2",
                  iSpeedOut=>"AO Скорость M2",
                  "rSpeedHMI(0-100)"=>"__MainBlock".Pump[2]."rHMI_Speed%",
                  bPumpRunning=>"__MainBlock".Pump[2].bHMI_RUN_State,
                  bPumpFault=>"__MainBlock".Pump[2].bALARM,
                  iStatus=>"__MainBlock".Pump[2].iHMI_Status);

   //Насос выхода из бочки М3
   "FB_Pump_DB_3"(bManualMode:="__MainBlock".Pump[3].bManualMode,
                  bManualStart:="__MainBlock".Pump[3].bManualStart,
                  bManualStop:=0,
                  rManualSpeed:="__MainBlock".Pump[3].rManualSpeed,
                  bDryRunn:= "fb_DI_LS1 - Низ Буфер",
                  bAutoSTop:=false,
                  bAutoStartPerm:="__MainBlock".Pump[3].bAutoCMD,
                  rAutoSpeed:="__MainBlock".Pump[3].rAutoSpeed,
                  bАвтоматы:=1,
                  bПускатели:=1,
                  bDriveRunning:="fb_DI_Работа ПЧ-3",
                  bDriveFault:=0,
                  rMinSpeed:=0.0,
                  rMaxSpeed:=100.0,
                  bResetFault:="__MainBlock".Pump[3].bResAlarm,
                  bRunCmd=>"Насос М3",
                  iSpeedOut=>"AO Скорость M3",
                  "rSpeedHMI(0-100)"=>"__MainBlock".Pump[3]."rHMI_Speed%",
                  bPumpRunning=>"__MainBlock".Pump[3].bHMI_RUN_State,
                  bPumpFault=>"__MainBlock".Pump[3].bALARM,
                  iStatus=>"__MainBlock".Pump[3].iHMI_Status);

   //Насос ГВС - подогрев М4
   "FB_Pump_DB_4"(bManualMode := "__MainBlock".Pump[4].bManualMode,
                  bManualStart := "__MainBlock".Pump[4].bManualStart,
                  bManualStop := 0,
                  rManualSpeed := "__MainBlock".Pump[4].rManualSpeed,
                  bDryRunn := 1,
                  bAutoSTop := false,
                  bAutoStartPerm := "__MainBlock".Pump[4].bAutoCMD,
                  rAutoSpeed := "__MainBlock".Pump[4].rAutoSpeed,
                  bАвтоматы := 1,
                  bПускатели := 1,
                  bDriveRunning := "fb_DI_Работа ПЧ-4",
                  bDriveFault := 0,
                  rMinSpeed := 0.0,
                  rMaxSpeed := 100.0,
                  bResetFault := "__MainBlock".Pump[4].bResAlarm,
                  bRunCmd => "Насос М4",
                  iSpeedOut => "AO Скорость M4",
                  "rSpeedHMI(0-100)" => "__MainBlock".Pump[4]."rHMI_Speed%",
                  bPumpRunning => "__MainBlock".Pump[4].bHMI_RUN_State,
                  bPumpFault => "__MainBlock".Pump[4].bALARM,
                  iStatus => "__MainBlock".Pump[4].iHMI_Status);


   //Насос защиты от перемерзания Гликоль М5
   "FB_Pump_DB_5"(bManualMode := "__MainBlock".Pump[5].bManualMode,
                  bManualStart := "__MainBlock".Pump[5].bManualStart,
                  bManualStop := 0,
                  rManualSpeed := "__MainBlock".Pump[5].rManualSpeed,
                  bDryRunn := 1,
                  bAutoSTop := false,
                  bAutoStartPerm := "__MainBlock".Pump[5].bAutoCMD,
                  rAutoSpeed := "__MainBlock".Pump[5].rAutoSpeed,
                  bАвтоматы := 1,
                  bПускатели := 1,
                  bDriveRunning := "fb_DI_Работа ПЧ-5",
                  bDriveFault := 0,
                  rMinSpeed := 0.0,
                  rMaxSpeed := 100.0,
                  bResetFault := "__MainBlock".Pump[5].bResAlarm,
                  bRunCmd => "Насос М5",
                  iSpeedOut => "AO Скорость M5",
                  "rSpeedHMI(0-100)" => "__MainBlock".Pump[5]."rHMI_Speed%",
                  bPumpRunning => "__MainBlock".Pump[5].bHMI_RUN_State,
                  bPumpFault => "__MainBlock".Pump[5].bALARM,
                  iStatus => "__MainBlock".Pump[5].iHMI_Status);
END_FUNCTION

FUNCTION "AI" : Void   // FC4, SCL
{ S7_Optimized_Access := 'TRUE' }
VERSION : 0.1
BEGIN

   "AI_Univ_DB_1"(iInValue:="AI TT1",                              //вход сигнала с датчика
                  iTypeSensor:="__MainBlock".AI[1].iTypeSensor,
                  bSimEnable:="__MainBlock".AI[1].bSimEnable,
                  rSimValue:="__MainBlock".AI[1].rSimValue,
                  rHL:="__MainBlock".AI[1].rHL,
                  rLL:="__MainBlock".AI[1].rLL,
                  bFilterEnable:="__MainBlock".AI[1].bFilterEnable,
                  rOut_Value=>"__MainBlock".AI[1].rOut_Value,
                  bOut_Error=>"__MainBlock".AI[1].bOut_Error);


   "AI_Univ_DB_2"(iInValue := "AI TT2",                            //вход сигнала с датчика
                  iTypeSensor := "__MainBlock".AI[2].iTypeSensor,
                  bSimEnable := "__MainBlock".AI[2].bSimEnable,
                  rSimValue := "__MainBlock".AI[2].rSimValue,
                  rHL := "__MainBlock".AI[2].rHL,
                  rLL := "__MainBlock".AI[2].rLL,
                  bFilterEnable := "__MainBlock".AI[2].bFilterEnable,
                  rOut_Value => "__MainBlock".AI[2].rOut_Value,
                  bOut_Error => "__MainBlock".AI[2].bOut_Error);


   "AI_Univ_DB_3"(iInValue := "AI TT3",                            //вход сигнала с датчика
                  iTypeSensor := "__MainBlock".AI[3].iTypeSensor,
                  bSimEnable := "__MainBlock".AI[3].bSimEnable,
                  rSimValue := "__MainBlock".AI[3].rSimValue,
                  rHL := "__MainBlock".AI[3].rHL,
                  rLL := "__MainBlock".AI[3].rLL,
                  bFilterEnable := "__MainBlock".AI[3].bFilterEnable,
                  rOut_Value => "__MainBlock".AI[3].rOut_Value,
                  bOut_Error => "__MainBlock".AI[3].bOut_Error);


   "AI_Univ_DB_4"(iInValue := "AI TT4",                            //вход сигнала с датчика
                  iTypeSensor := "__MainBlock".AI[4].iTypeSensor,
                  bSimEnable := "__MainBlock".AI[4].bSimEnable,
                  rSimValue := "__MainBlock".AI[4].rSimValue,
                  rHL := "__MainBlock".AI[4].rHL,
                  rLL := "__MainBlock".AI[4].rLL,
                  bFilterEnable := "__MainBlock".AI[4].bFilterEnable,
                  rOut_Value => "__MainBlock".AI[4].rOut_Value,
                  bOut_Error => "__MainBlock".AI[4].bOut_Error);

   "AI_Univ_DB_5"(iInValue := "AI TT5",                            //вход сигнала с датчика
                  iTypeSensor := "__MainBlock".AI[5].iTypeSensor,
                  bSimEnable := "__MainBlock".AI[5].bSimEnable,
                  rSimValue := "__MainBlock".AI[5].rSimValue,
                  rHL := "__MainBlock".AI[5].rHL,
                  rLL := "__MainBlock".AI[5].rLL,
                  bFilterEnable := "__MainBlock".AI[5].bFilterEnable,
                  rOut_Value => "__MainBlock".AI[5].rOut_Value,
                  bOut_Error => "__MainBlock".AI[5].bOut_Error);


   "AI_Univ_DB_6"(iInValue := "AI TT6",                            //вход сигнала с датчика
                  iTypeSensor := "__MainBlock".AI[6].iTypeSensor,
                  bSimEnable := "__MainBlock".AI[6].bSimEnable,
                  rSimValue := "__MainBlock".AI[6].rSimValue,
                  rHL := "__MainBlock".AI[6].rHL,
                  rLL := "__MainBlock".AI[6].rLL,
                  bFilterEnable := "__MainBlock".AI[6].bFilterEnable,
                  rOut_Value => "__MainBlock".AI[6].rOut_Value,
                  bOut_Error => "__MainBlock".AI[6].bOut_Error);

   "AI_Univ_DB_7"(iInValue := "AI Расходомерр",                            //вход сигнала с датчика
                  iTypeSensor := "__MainBlock".AI[7].iTypeSensor,
                  bSimEnable := "__MainBlock".AI[7].bSimEnable,
                  rSimValue := "__MainBlock".AI[7].rSimValue,
                  rHL := "__MainBlock".AI[7].rHL,
                  rLL := "__MainBlock".AI[7].rLL,
                  bFilterEnable := "__MainBlock".AI[7].bFilterEnable,
                  rOut_Value => "__MainBlock".AI[7].rOut_Value,
                  bOut_Error => "__MainBlock".AI[7].bOut_Error);


   "AI_Univ_DB_8"(iInValue := "AI PT1",                            //вход сигнала с датчика
                  iTypeSensor := "__MainBlock".AI[8].iTypeSensor,
                  bSimEnable := "__MainBlock".AI[8].bSimEnable,
                  rSimValue := "__MainBlock".AI[8].rSimValue,
                  rHL := "__MainBlock".AI[8].rHL,
                  rLL := "__MainBlock".AI[8].rLL,
                  bFilterEnable := "__MainBlock".AI[8].bFilterEnable,
                  rOut_Value => "__MainBlock".AI[8].rOut_Value,
                  bOut_Error => "__MainBlock".AI[8].bOut_Error);

   "AI_Univ_DB_9"(iInValue := "AI PT2 - Секция пастеризации",                            //вход сигнала с датчикадаление секции пастеризации
                  iTypeSensor := "__MainBlock".AI[9].iTypeSensor,
                  bSimEnable := "__MainBlock".AI[9].bSimEnable,
                  rSimValue := "__MainBlock".AI[9].rSimValue,
                  rHL := "__MainBlock".AI[9].rHL,
                  rLL := "__MainBlock".AI[9].rLL,
                  bFilterEnable := "__MainBlock".AI[9].bFilterEnable,
                  rOut_Value => "__MainBlock".AI[9].rOut_Value,
                  bOut_Error => "__MainBlock".AI[9].bOut_Error);


   "AI_Univ_DB_10"(iInValue := "AI PT3",                            //вход сигнала с датчика
                   iTypeSensor := "__MainBlock".AI[10].iTypeSensor,
                   bSimEnable := "__MainBlock".AI[10].bSimEnable,
                   rSimValue := "__MainBlock".AI[10].rSimValue,
                   rHL := "__MainBlock".AI[10].rHL,
                   rLL := "__MainBlock".AI[10].rLL,
                   bFilterEnable := "__MainBlock".AI[10].bFilterEnable,
                   rOut_Value => "__MainBlock".AI[10].rOut_Value,
                   bOut_Error => "__MainBlock".AI[10].bOut_Error);

   "AI_Univ_DB_11"(iInValue := "AI WT",                            //вход сигнала с датчика
                   iTypeSensor := "__MainBlock".AI[11].iTypeSensor,
                   bSimEnable := "__MainBlock".AI[11].bSimEnable,
                   rSimValue := "__MainBlock".AI[11].rSimValue,
                   rHL := "__MainBlock".AI[11].rHL,
                   rLL := "__MainBlock".AI[11].rLL,
                   bFilterEnable := "__MainBlock".AI[11].bFilterEnable,
                   rOut_Value => "__MainBlock".AI[11].rOut_Value,
                   bOut_Error => "__MainBlock".AI[11].bOut_Error);

   "AI_Univ_DB_12"(iInValue := "AI CT",                            //вход сигнала с датчика
                   iTypeSensor := "__MainBlock".AI[12].iTypeSensor,
                   bSimEnable := "__MainBlock".AI[12].bSimEnable,
                   rSimValue := "__MainBlock".AI[12].rSimValue,
                   rHL := "__MainBlock".AI[12].rHL,
                   rLL := "__MainBlock".AI[12].rLL,
                   bFilterEnable := "__MainBlock".AI[12].bFilterEnable,
                   rOut_Value => "__MainBlock".AI[12].rOut_Value,
                   bOut_Error => "__MainBlock".AI[12].bOut_Error);


   //для читаемости кода можно использовать как массивные данные так и именнованные для HMI
   //
   "fb_AI_Темп входа пива PT100" :=          "__MainBlock".AI[1].rOut_Value;
   "fb_AI_Темп выхода пива  PT100" :=        "__MainBlock".AI[2].rOut_Value;
   "fb_AI_Темп ГВ - нагрев PT100" :=         "__MainBlock".AI[3].rOut_Value;
   "fb_AI_Темп Гликоль PT100" :=             "__MainBlock".AI[4].rOut_Value;
   "fb_AI_ТЕмп емкость PT100" :=             "__MainBlock".AI[5].rOut_Value;
   "fb_AI_Темп выход продукт ТТ6 4-20 мА" := "__MainBlock".AI[6].rOut_Value;
   "Расход ПОУ" :=                           "__MainBlock".AI[7].rOut_Value;
   "fb_AI_M2_давления 4-20" :=               "__MainBlock".AI[8].rOut_Value;
   "fb_AI_Выход пива давления 4-20" :=       "__MainBlock".AI[9].rOut_Value;
   "fb_AI_Выход Буфера давления 4-20" :=     "__MainBlock".AI[10].rOut_Value;
   "fb_AI_Датчик веса буфера" :=             "__MainBlock".AI[11].rOut_Value;
   "fb_AI_Датчик концентрации" :=            "__MainBlock".AI[12].rOut_Value;
END_FUNCTION

FUNCTION "FC_Valve_o/c" : Void   // FC5, SCL
{ S7_Optimized_Access := 'TRUE' }
VERSION : 0.1
BEGIN

   //........................Присваиваем обработанный сигнал входа статуса открытия клапана к входу блока обработки клапана//........................
   //
   "__MainBlock"."Valve_o/c"[1].bFeedbackOpen := NOT "fb_DI_Состояние V1";
   "__MainBlock"."Valve_o/c"[2].bFeedbackOpen := NOT "fb_DI_Состояние V2";
   "__MainBlock"."Valve_o/c"[3].bFeedbackOpen := "fb_DI_Состояние V3";
   "__MainBlock"."Valve_o/c"[4].bFeedbackOpen := NOT "fb_DI_Состояние V4";
   "__MainBlock"."Valve_o/c"[5].bFeedbackOpen := NOT "fb_DI_Состояние V5";
   "__MainBlock"."Valve_o/c"[6].bFeedbackOpen := NOT "fb_DI_Состояние V6";
   "__MainBlock"."Valve_o/c"[7].bFeedbackOpen := NOT "fb_DI_Состояние V7";
   "__MainBlock"."Valve_o/c"[8].bFeedbackOpen := NOT "fb_DI_Состояние V8";
   "__MainBlock"."Valve_o/c"[9].bFeedbackOpen := NOT "fb_DI_Состояние V9";
   "__MainBlock"."Valve_o/c"[10].bFeedbackOpen := "fb_DI_Состояние V10";
   // ................................................................................................................................................


   //Передача данных в ФБ обработки



   "Valve_o/c_fb_Arrey_old_DB"("__MainBlock"."Valve_o/c");


   //........................Присваиваем обработанный выход к физическим выходам модуля...............................................................

   "V1_Вода" :=                "__MainBlock"."Valve_o/c"[1].bValveOut;
   "V2_Продукт" :=             "__MainBlock"."Valve_o/c"[2].bValveOut;
   "V3_Давления" :=            "__MainBlock"."Valve_o/c"[3].bValveOut;
   "V4_Циркуляция" :=          "__MainBlock"."Valve_o/c"[4].bValveOut;
   "V5_Дренаж (НО)" :=         "__MainBlock"."Valve_o/c"[5].bValveOut;
   "V6_Возврат" :=             "__MainBlock"."Valve_o/c"[6].bValveOut;
   "V7_Моющая головка" :=      "__MainBlock"."Valve_o/c"[7].bValveOut;
   "V8_Вход пр в бочку" :=     "__MainBlock"."Valve_o/c"[8].bValveOut;
   "V9_Выход пр из бочки" :=   "__MainBlock"."Valve_o/c"[9].bValveOut;
   "V10_клапан" :=             "__MainBlock"."Valve_o/c"[10].bValveOut;
   "V11_Запорный тепло" :=     "__MainBlock"."Valve_o/c"[11].bValveOut;
   "V12_Запор гликоль" :=      "__MainBlock"."Valve_o/c"[12].bValveOut;
   "V13_Сброс дав емкость" :=  "__MainBlock"."Valve_o/c"[13].bValveOut;
   "V14_Щелочь" :=             "__MainBlock"."Valve_o/c"[14].bValveOut;
   "V15_Насос Щелочь" :=       "__MainBlock"."Valve_o/c"[15].bValveOut;
   "V16_Кислота" :=            "__MainBlock"."Valve_o/c"[16].bValveOut;
   "V17_Насос Кислота" :=      "__MainBlock"."Valve_o/c"[17].bValveOut;
END_FUNCTION

FUNCTION "Аварии/res" : Void   // FC6, LAD
{ S7_Optimized_Access := 'TRUE' }
VERSION : 0.1
   VAR_INPUT
      bResrt : Bool;
   END_VAR
   VAR_OUTPUT
      xAlarm : Bool;   // Есть активные аварии
   END_VAR
BEGIN

REGION Network 1
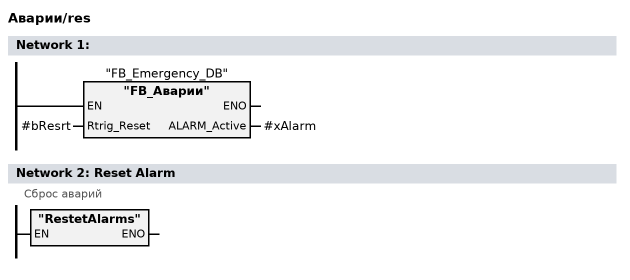
   RUNG wire#powerrail
      "FB_Emergency_DB"(Rtrig_Reset := #bResrt, ALARM_Active => #xAlarm)
   END_RUNG
   // the same network as SCL:
   "FB_Emergency_DB"(Rtrig_Reset := #bResrt, ALARM_Active => #xAlarm);   // "FB_Аварии"
END_REGION

REGION Network 2: Reset Alarm
   // Сброс аварий
   RUNG wire#powerrail
      "RestetAlarms"()
   END_RUNG
   // the same network as SCL:
   "RestetAlarms"();
END_REGION

REGION Network 3 (SCL): Есть активные аварии
END_REGION
END_FUNCTION

FUNCTION "FC_Valve-Regul" : Void   // FC8, SCL
{ S7_Optimized_Access := 'TRUE' }
VERSION : 0.1
BEGIN
   //========================================== ВХОДЫ  =============================================================
   //сМОТРИ ПИД

   "__MainBlock".Valve_Regul[1].rAutoSetpoint := "iPID_Out_Нагрев";
   "__MainBlock".Valve_Regul[2].rAutoSetpoint := "iPID_Out_Гликоль";
   "__MainBlock".Valve_Regul[3].rAutoSetpoint := "iPID_Out_Кл.Давления";
   "__MainBlock".Valve_Regul[3].bAutoOpenClose := "__MainBlock"."Valve_o/c"[3].bAuto_OpenCmd;



   //
   //Передача данных в ФБ обработки

   "fb_Valve-regul_DB"("__MainBlock".Valve_Regul);


   //========================================== ВЫХОДА  =============================================================

